LIN {X 0,Y 505.986,Z 301.18,A -85,B 0,C 180,E1 23907.931,E2 23907.931} C_VEL
LIN {X 0,Y 499.705,Z 283.022,A -85,B 0,C 180,E1 23905.729,E2 23905.729} C_VEL
LIN {X 0,Y 496.793,Z 274.791,A -85,B 0,C 180,E1 23904.638,E2 23904.638} C_VEL
LIN {X 0,Y 496.772,Z 274.605,A -85,B 0,C 180,E1 23901.099,E2 23901.099} C_VEL
LIN {X 0,Y 496.748,Z 274.605,A -85,B 0,C 180,E1 23897.6,E2 23897.6} C_VEL
LIN {X 0,Y 496.751,Z 274.607,A -85,B 0,C 180,E1 23893.982,E2 23893.982} C_VEL
LIN {X 0,Y 496.769,Z 274.603,A -85,B 0,C 180,E1 23890.399,E2 23890.399} C_VEL
LIN {X 0,Y 496.757,Z 274.604,A -85,B 0,C 180,E1 23886.857,E2 23886.857} C_VEL
LIN {X 0,Y 496.761,Z 274.607,A -85,B 0,C 180,E1 23883.333,E2 23883.333} C_VEL
LIN {X 0,Y 496.769,Z 274.598,A -85,B 0,C 180,E1 23879.812,E2 23879.812} C_VEL
LIN {X 0,Y 496.768,Z 274.604,A -85,B 0,C 180,E1 23876.284,E2 23876.284} C_VEL
LIN {X 0,Y 496.734,Z 274.607,A -85,B 0,C 180,E1 23872.794,E2 23872.794} C_VEL
LIN {X 0,Y 496.727,Z 274.609,A -85,B 0,C 180,E1 23869.255,E2 23869.255} C_VEL
LIN {X 0,Y 496.753,Z 274.6,A -85,B 0,C 180,E1 23865.768,E2 23865.768} C_VEL
LIN {X 0,Y 496.743,Z 274.605,A -85,B 0,C 180,E1 23862.32,E2 23862.32} C_VEL
LIN {X 0,Y 496.744,Z 274.899,A -85,B 0,C 180,E1 23861.172,E2 23861.172} C_VEL
LIN {X 0,Y 503.539,Z 295.552,A -85,B 0,C 180,E1 23858.969,E2 23858.969} C_VEL
LIN {X 0,Y 503.974,Z 298.794,A -85,B 0,C 180,E1 23858.673,E2 23858.673} C_VEL
LIN {X 0,Y 503.208,Z 340.602,A -85,B 0,C 180,E1 23855.245,E2 23855.245} C_VEL
LIN {X 0,Y 502.249,Z 380.984,A -85,B 0,C 180,E1 23851.941,E2 23851.941} C_VEL
LIN {X 0,Y 501.067,Z 425.768,A -85,B 0,C 180,E1 23848.286,E2 23848.286} C_VEL
LIN {X 0,Y 500.006,Z 468.043,A -85,B 0,C 180,E1 23844.839,E2 23844.839} C_VEL
LIN {X 0,Y 499.903,Z 474.861,A -85,B 0,C 180,E1 23844.316,E2 23844.316} C_VEL
LIN {X 0,Y 500.969,Z 485.924,A -85,B 0,C 180,E1 23844.105,E2 23844.105} C_VEL
LIN {X 0,Y 499.941,Z 617.34,A -85,B 0,C 180,E1 23842.16,E2 23842.16} C_VEL
LIN {X 0,Y 499.655,Z 633.277,A -85,B 0,C 180,E1 23841.714,E2 23841.714} C_VEL
LIN {X 0,Y 499.205,Z 649.81,A -85,B 0,C 180,E1 23841.013,E2 23841.013} C_VEL
LIN {X 0,Y 498.696,Z 664.017,A -85,B 0,C 180,E1 23840.189,E2 23840.189} C_VEL
LIN {X 0,Y 498.107,Z 678.224,A -85,B 0,C 180,E1 23839.125,E2 23839.125} C_VEL
LIN {X 0,Y 497.578,Z 690.76,A -85,B 0,C 180,E1 23837.939,E2 23837.939} C_VEL
LIN {X 0,Y 497.048,Z 702.83,A -85,B 0,C 180,E1 23836.507,E2 23836.507} C_VEL
LIN {X 0,Y 496.653,Z 712.568,A -85,B 0,C 180,E1 23835.069,E2 23835.069} C_VEL
LIN {X 0,Y 496.323,Z 721.598,A -85,B 0,C 180,E1 23833.379,E2 23833.379} C_VEL
LIN {X 0,Y 496.123,Z 728.676,A -85,B 0,C 180,E1 23831.666,E2 23831.666} C_VEL
LIN {X 0,Y 496.01,Z 734.174,A -85,B 0,C 180,E1 23829.838,E2 23829.838} C_VEL
LIN {X 0,Y 495.963,Z 737.914,A -85,B 0,C 180,E1 23827.979,E2 23827.979} C_VEL
LIN {X 0,Y 495.946,Z 739.841,A -85,B 0,C 180,E1 23826.096,E2 23826.096} C_VEL
LIN {X 0,Y 495.945,Z 740.052,A -85,B 0,C 180,E1 23824.187,E2 23824.187} C_VEL
LIN {X 0,Y 495.956,Z 738.355,A -85,B 0,C 180,E1 23822.246,E2 23822.246} C_VEL
LIN {X 0,Y 496.004,Z 734.845,A -85,B 0,C 180,E1 23820.323,E2 23820.323} C_VEL
LIN {X 0,Y 496.106,Z 729.548,A -85,B 0,C 180,E1 23818.488,E2 23818.488} C_VEL
LIN {X 0,Y 496.302,Z 722.599,A -85,B 0,C 180,E1 23816.728,E2 23816.728} C_VEL
LIN {X 0,Y 496.624,Z 713.491,A -85,B 0,C 180,E1 23814.987,E2 23814.987} C_VEL
LIN {X 0,Y 497.041,Z 703.344,A -85,B 0,C 180,E1 23813.458,E2 23813.458} C_VEL
LIN {X 0,Y 497.549,Z 691.637,A -85,B 0,C 180,E1 23812.056,E2 23812.056} C_VEL
LIN {X 0,Y 498.077,Z 679.489,A -85,B 0,C 180,E1 23810.881,E2 23810.881} C_VEL
LIN {X 0,Y 498.659,Z 665.144,A -85,B 0,C 180,E1 23809.789,E2 23809.789} C_VEL
LIN {X 0,Y 499.193,Z 650.674,A -85,B 0,C 180,E1 23808.933,E2 23808.933} C_VEL
LIN {X 0,Y 499.631,Z 634.514,A -85,B 0,C 180,E1 23808.237,E2 23808.237} C_VEL
LIN {X 0,Y 499.922,Z 618.388,A -85,B 0,C 180,E1 23807.769,E2 23807.769} C_VEL
LIN {X 0,Y 500.3,Z 568.29,A -85,B 0,C 180,E1 23807.005,E2 23807.005} C_VEL
LIN {X 0,Y 500.781,Z 482.143,A -85,B 0,C 180,E1 23805.739,E2 23805.739} C_VEL
LIN {X 0,Y 499.842,Z 474.397,A -85,B 0,C 180,E1 23805.566,E2 23805.566} C_VEL
LIN {X 0,Y 500.963,Z 429.094,A -85,B 0,C 180,E1 23801.89,E2 23801.89} C_VEL
LIN {X 0,Y 501.829,Z 393.421,A -85,B 0,C 180,E1 23799.012,E2 23799.012} C_VEL
LIN {X 0,Y 502.557,Z 361.365,A -85,B 0,C 180,E1 23796.433,E2 23796.433} C_VEL
LIN {X 0,Y 503.208,Z 320.138,A -85,B 0,C 180,E1 23793.122,E2 23793.122} C_VEL
LIN {X 0,Y 503.4,Z 295.62,A -85,B 0,C 180,E1 23791.159,E2 23791.159} C_VEL
LIN {X 0,Y 496.791,Z 274.932,A -85,B 0,C 180,E1 23789.049,E2 23789.049} C_VEL
LIN {X 0,Y 496.729,Z 274.611,A -85,B 0,C 180,E1 23788.363,E2 23788.363} C_VEL
LIN {X 0,Y 496.731,Z 274.611,A -85,B 0,C 180,E1 23784.752,E2 23784.752} C_VEL
LIN {X 0,Y 496.766,Z 274.602,A -85,B 0,C 180,E1 23781.242,E2 23781.242} C_VEL
LIN {X 0,Y 496.764,Z 274.605,A -85,B 0,C 180,E1 23777.694,E2 23777.694} C_VEL
LIN {X 0,Y 496.729,Z 274.608,A -85,B 0,C 180,E1 23774.216,E2 23774.216} C_VEL
LIN {X 0,Y 496.736,Z 274.605,A -85,B 0,C 180,E1 23770.672,E2 23770.672} C_VEL
LIN {X 0,Y 496.774,Z 274.603,A -85,B 0,C 180,E1 23767.148,E2 23767.148} C_VEL
LIN {X 0,Y 496.764,Z 274.607,A -85,B 0,C 180,E1 23763.578,E2 23763.578} C_VEL
LIN {X 0,Y 496.733,Z 274.608,A -85,B 0,C 180,E1 23760.116,E2 23760.116} C_VEL
LIN {X 0,Y 496.738,Z 274.604,A -85,B 0,C 180,E1 23756.538,E2 23756.538} C_VEL
LIN {X 0,Y 496.773,Z 274.603,A -85,B 0,C 180,E1 23753.064,E2 23753.064} C_VEL
LIN {X 0,Y 496.757,Z 274.606,A -85,B 0,C 180,E1 23749.564,E2 23749.564} C_VEL
LIN {X 0,Y 496.734,Z 274.606,A -85,B 0,C 180,E1 23746.023,E2 23746.023} C_VEL
LIN {X 0,Y 496.744,Z 274.605,A -85,B 0,C 180,E1 23742.427,E2 23742.427} C_VEL
LIN {X 0,Y 496.771,Z 274.602,A -85,B 0,C 180,E1 23738.883,E2 23738.883} C_VEL
LIN {X 0,Y 496.763,Z 274.607,A -85,B 0,C 180,E1 23735.378,E2 23735.378} C_VEL
LIN {X 0,Y 496.738,Z 274.607,A -85,B 0,C 180,E1 23731.835,E2 23731.835} C_VEL
LIN {X 0,Y 496.746,Z 274.603,A -85,B 0,C 180,E1 23728.309,E2 23728.309} C_VEL
LIN {X 0,Y 496.772,Z 274.604,A -85,B 0,C 180,E1 23724.798,E2 23724.798} C_VEL
LIN {X 0,Y 496.767,Z 274.609,A -85,B 0,C 180,E1 23721.248,E2 23721.248} C_VEL
LIN {X 0,Y 496.739,Z 274.609,A -85,B 0,C 180,E1 23717.756,E2 23717.756} C_VEL
LIN {X 0,Y 496.751,Z 274.605,A -85,B 0,C 180,E1 23714.23,E2 23714.23} C_VEL
LIN {X 0,Y 496.772,Z 274.607,A -85,B 0,C 180,E1 23710.699,E2 23710.699} C_VEL
LIN {X 0,Y 496.777,Z 274.865,A -85,B 0,C 180,E1 23707.944,E2 23707.944} C_VEL
LIN {X 0,Y 500.523,Z 284.291,A -85,B 0,C 180,E1 23706.77,E2 23706.77} C_VEL
LIN {X 0,Y 508.094,Z 303.988,A -85,B 0,C 180,E1 23704.559,E2 23704.559} C_VEL
LIN {X 0,Y 507.57,Z 316.675,A -85,B 0,C 180,E1 23703.616,E2 23703.616} C_VEL
LIN {X 0,Y 510.176,Z 334.45,A -85,B 0,C 180,E1 23703.112,E2 23703.112} C_VEL
LIN {X 0,Y 508.469,Z 453.813,A -85,B 0,C 180,E1 23701.237,E2 23701.237} C_VEL
LIN {X 0,Y 506.934,Z 577.933,A -85,B 0,C 180,E1 23699.32,E2 23699.32} C_VEL
LIN {X 0,Y 506.225,Z 599.572,A -85,B 0,C 180,E1 23698.769,E2 23698.769} C_VEL
LIN {X 0,Y 505.38,Z 619.891,A -85,B 0,C 180,E1 23698.031,E2 23698.031} C_VEL
LIN {X 0,Y 504.378,Z 639.254,A -85,B 0,C 180,E1 23697.117,E2 23697.117} C_VEL
LIN {X 0,Y 503.262,Z 658.557,A -85,B 0,C 180,E1 23695.981,E2 23695.981} C_VEL
LIN {X 0,Y 502.09,Z 677.202,A -85,B 0,C 180,E1 23694.641,E2 23694.641} C_VEL
LIN {X 0,Y 500.925,Z 694.485,A -85,B 0,C 180,E1 23693.153,E2 23693.153} C_VEL
LIN {X 0,Y 499.847,Z 710.302,A -85,B 0,C 180,E1 23691.542,E2 23691.542} C_VEL
LIN {X 0,Y 498.832,Z 724.453,A -85,B 0,C 180,E1 23689.799,E2 23689.799} C_VEL
LIN {X 0,Y 497.924,Z 737.789,A -85,B 0,C 180,E1 23687.859,E2 23687.859} C_VEL
LIN {X 0,Y 497.213,Z 749.382,A -85,B 0,C 180,E1 23685.87,E2 23685.87} C_VEL
LIN {X 0,Y 496.65,Z 760.337,A -85,B 0,C 180,E1 23683.622,E2 23683.622} C_VEL
LIN {X 0,Y 496.279,Z 769.255,A -85,B 0,C 180,E1 23681.386,E2 23681.386} C_VEL
LIN {X 0,Y 496.067,Z 776.378,A -85,B 0,C 180,E1 23679.161,E2 23679.161} C_VEL
LIN {X 0,Y 495.965,Z 782.008,A -85,B 0,C 180,E1 23676.83,E2 23676.83} C_VEL
LIN {X 0,Y 495.918,Z 785.929,A -85,B 0,C 180,E1 23674.509,E2 23674.509} C_VEL
LIN {X 0,Y 495.911,Z 788.305,A -85,B 0,C 180,E1 23672.079,E2 23672.079} C_VEL
LIN {X 0,Y 495.906,Z 788.962,A -85,B 0,C 180,E1 23669.768,E2 23669.768} C_VEL
LIN {X 0,Y 495.908,Z 788.03,A -85,B 0,C 180,E1 23667.456,E2 23667.456} C_VEL
LIN {X 0,Y 495.924,Z 785.445,A -85,B 0,C 180,E1 23665.141,E2 23665.141} C_VEL
LIN {X 0,Y 495.964,Z 781.241,A -85,B 0,C 180,E1 23662.819,E2 23662.819} C_VEL
LIN {X 0,Y 496.095,Z 775.322,A -85,B 0,C 180,E1 23660.486,E2 23660.486} C_VEL
LIN {X 0,Y 496.335,Z 767.956,A -85,B 0,C 180,E1 23658.247,E2 23658.247} C_VEL
LIN {X 0,Y 496.733,Z 758.589,A -85,B 0,C 180,E1 23655.977,E2 23655.977} C_VEL
LIN {X 0,Y 497.288,Z 748.099,A -85,B 0,C 180,E1 23653.89,E2 23653.89} C_VEL
LIN {X 0,Y 498.033,Z 736.03,A -85,B 0,C 180,E1 23651.869,E2 23651.869} C_VEL
LIN {X 0,Y 499.023,Z 721.655,A -85,B 0,C 180,E1 23649.84,E2 23649.84} C_VEL
LIN {X 0,Y 500.037,Z 707.603,A -85,B 0,C 180,E1 23648.165,E2 23648.165} C_VEL
LIN {X 0,Y 501.074,Z 691.666,A -85,B 0,C 180,E1 23646.603,E2 23646.603} C_VEL
LIN {X 0,Y 502.192,Z 674.015,A -85,B 0,C 180,E1 23645.158,E2 23645.158} C_VEL
LIN {X 0,Y 503.256,Z 655.481,A -85,B 0,C 180,E1 23643.899,E2 23643.899} C_VEL
LIN {X 0,Y 504.197,Z 636.876,A -85,B 0,C 180,E1 23642.863,E2 23642.863} C_VEL
LIN {X 0,Y 505.11,Z 616.417,A -85,B 0,C 180,E1 23641.956,E2 23641.956} C_VEL
LIN {X 0,Y 505.853,Z 595.464,A -85,B 0,C 180,E1 23641.258,E2 23641.258} C_VEL
LIN {X 0,Y 506.394,Z 574.481,A -85,B 0,C 180,E1 23640.774,E2 23640.774} C_VEL
LIN {X 0,Y 508.288,Z 392.914,A -85,B 0,C 180,E1 23638.038,E2 23638.038} C_VEL
LIN {X 0,Y 509.019,Z 331.819,A -85,B 0,C 180,E1 23637.033,E2 23637.033} C_VEL
LIN {X 0,Y 506.9,Z 317.552,A -85,B 0,C 180,E1 23636.61,E2 23636.61} C_VEL
LIN {X 0,Y 507.597,Z 303.416,A -85,B 0,C 180,E1 23635.523,E2 23635.523} C_VEL
LIN {X 0,Y 501.679,Z 286.882,A -85,B 0,C 180,E1 23633.563,E2 23633.563} C_VEL
LIN {X 0,Y 498.35,Z 278.58,A -85,B 0,C 180,E1 23632.415,E2 23632.415} C_VEL
LIN {X 0,Y 496.787,Z 274.85,A -85,B 0,C 180,E1 23631.796,E2 23631.796} C_VEL
LIN {X 0,Y 496.734,Z 274.612,A -85,B 0,C 180,E1 23628.311,E2 23628.311} C_VEL
LIN {X 0,Y 496.754,Z 274.611,A -85,B 0,C 180,E1 23624.787,E2 23624.787} C_VEL
LIN {X 0,Y 496.775,Z 274.607,A -85,B 0,C 180,E1 23621.312,E2 23621.312} C_VEL
LIN {X 0,Y 496.735,Z 274.612,A -85,B 0,C 180,E1 23617.873,E2 23617.873} C_VEL
LIN {X 0,Y 496.768,Z 274.901,A -85,B 0,C 180,E1 23616.1,E2 23616.1} C_VEL
LIN {X 0,Y 500.068,Z 282.968,A -85,B 0,C 180,E1 23614.736,E2 23614.736} C_VEL
LIN {X 0,Y 504.417,Z 294.778,A -85,B 0,C 180,E1 23613.032,E2 23613.032} C_VEL
LIN {X 0,Y 506.659,Z 302.39,A -85,B 0,C 180,E1 23612.063,E2 23612.063} C_VEL
LIN {X 0,Y 504.302,Z 341.082,A -85,B 0,C 180,E1 23608.577,E2 23608.577} C_VEL
LIN {X 0,Y 507.189,Z 359.883,A -85,B 0,C 180,E1 23608.008,E2 23608.008} C_VEL
LIN {X 0,Y 505.208,Z 474.152,A -85,B 0,C 180,E1 23606.152,E2 23606.152} C_VEL
LIN {X 0,Y 504.179,Z 561.011,A -85,B 0,C 180,E1 23604.803,E2 23604.803} C_VEL
LIN {X 0,Y 503.6,Z 581.084,A -85,B 0,C 180,E1 23604.273,E2 23604.273} C_VEL
LIN {X 0,Y 502.863,Z 599.834,A -85,B 0,C 180,E1 23603.556,E2 23603.556} C_VEL
LIN {X 0,Y 501.968,Z 618.446,A -85,B 0,C 180,E1 23602.608,E2 23602.608} C_VEL
LIN {X 0,Y 501.011,Z 635.928,A -85,B 0,C 180,E1 23601.482,E2 23601.482} C_VEL
LIN {X 0,Y 500.015,Z 652.165,A -85,B 0,C 180,E1 23600.178,E2 23600.178} C_VEL
LIN {X 0,Y 498.991,Z 668.376,A -85,B 0,C 180,E1 23598.596,E2 23598.596} C_VEL
LIN {X 0,Y 498.163,Z 681.6,A -85,B 0,C 180,E1 23597.039,E2 23597.039} C_VEL
LIN {X 0,Y 497.426,Z 694.289,A -85,B 0,C 180,E1 23595.267,E2 23595.267} C_VEL
LIN {X 0,Y 496.85,Z 705.515,A -85,B 0,C 180,E1 23593.381,E2 23593.381} C_VEL
LIN {X 0,Y 496.427,Z 715.203,A -85,B 0,C 180,E1 23591.384,E2 23591.384} C_VEL
LIN {X 0,Y 496.162,Z 722.983,A -85,B 0,C 180,E1 23589.394,E2 23589.394} C_VEL
LIN {X 0,Y 496.006,Z 729.436,A -85,B 0,C 180,E1 23587.296,E2 23587.296} C_VEL
LIN {X 0,Y 495.94,Z 734.373,A -85,B 0,C 180,E1 23585.089,E2 23585.089} C_VEL
LIN {X 0,Y 495.914,Z 737.458,A -85,B 0,C 180,E1 23582.889,E2 23582.889} C_VEL
LIN {X 0,Y 495.914,Z 738.85,A -85,B 0,C 180,E1 23580.693,E2 23580.693} C_VEL
LIN {X 0,Y 495.91,Z 738.609,A -85,B 0,C 180,E1 23578.498,E2 23578.498} C_VEL
LIN {X 0,Y 495.912,Z 736.657,A -85,B 0,C 180,E1 23576.3,E2 23576.3} C_VEL
LIN {X 0,Y 495.949,Z 732.923,A -85,B 0,C 180,E1 23574.098,E2 23574.098} C_VEL
LIN {X 0,Y 496.049,Z 727.391,A -85,B 0,C 180,E1 23571.888,E2 23571.888} C_VEL
LIN {X 0,Y 496.238,Z 720.359,A -85,B 0,C 180,E1 23569.786,E2 23569.786} C_VEL
LIN {X 0,Y 496.56,Z 711.892,A -85,B 0,C 180,E1 23567.794,E2 23567.794} C_VEL
LIN {X 0,Y 497.034,Z 701.633,A -85,B 0,C 180,E1 23565.842,E2 23565.842} C_VEL
LIN {X 0,Y 497.658,Z 690.096,A -85,B 0,C 180,E1 23564.023,E2 23564.023} C_VEL
LIN {X 0,Y 498.427,Z 677.376,A -85,B 0,C 180,E1 23562.34,E2 23562.34} C_VEL
LIN {X 0,Y 499.319,Z 663.137,A -85,B 0,C 180,E1 23560.767,E2 23560.767} C_VEL
LIN {X 0,Y 500.335,Z 646.924,A -85,B 0,C 180,E1 23559.285,E2 23559.285} C_VEL
LIN {X 0,Y 501.337,Z 630.264,A -85,B 0,C 180,E1 23558.033,E2 23558.033} C_VEL
LIN {X 0,Y 502.287,Z 612.613,A -85,B 0,C 180,E1 23556.973,E2 23556.973} C_VEL
LIN {X 0,Y 503.176,Z 593.403,A -85,B 0,C 180,E1 23556.074,E2 23556.074} C_VEL
LIN {X 0,Y 503.874,Z 574.138,A -85,B 0,C 180,E1 23555.411,E2 23555.411} C_VEL
LIN {X 0,Y 504.363,Z 554.443,A -85,B 0,C 180,E1 23554.966,E2 23554.966} C_VEL
LIN {X 0,Y 506.641,Z 358.228,A -85,B 0,C 180,E1 23551.968,E2 23551.968} C_VEL
LIN {X 0,Y 505.059,Z 353.42,A -85,B 0,C 180,E1 23551.781,E2 23551.781} C_VEL
LIN {X 0,Y 499.919,Z 345.851,A -85,B 0,C 180,E1 23551.315,E2 23551.315} C_VEL
LIN {X 0,Y 497.214,Z 341.288,A -85,B 0,C 180,E1 23550.985,E2 23550.985} C_VEL
LIN {X 0,Y 496.832,Z 338.92,A -85,B 0,C 180,E1 23550.787,E2 23550.787} C_VEL
LIN {X 0,Y 498.75,Z 303.753,A -85,B 0,C 180,E1 23547.638,E2 23547.638} C_VEL
LIN {X 0,Y 491.879,Z 284.216,A -85,B 0,C 180,E1 23545.209,E2 23545.209} C_VEL
LIN {X 0,Y 488.822,Z 275.791,A -85,B 0,C 180,E1 23544.059,E2 23544.059} C_VEL
LIN {X 0,Y 488.834,Z 275.59,A -85,B 0,C 180,E1 23540.64,E2 23540.64} C_VEL
LIN {X 0,Y 488.83,Z 275.597,A -85,B 0,C 180,E1 23537.068,E2 23537.068} C_VEL
LIN {X 0,Y 488.823,Z 275.593,A -85,B 0,C 180,E1 23533.436,E2 23533.436} C_VEL
LIN {X 0,Y 488.818,Z 275.596,A -85,B 0,C 180,E1 23529.91,E2 23529.91} C_VEL
LIN {X 0,Y 488.828,Z 275.591,A -85,B 0,C 180,E1 23526.302,E2 23526.302} C_VEL
LIN {X 0,Y 488.814,Z 275.593,A -85,B 0,C 180,E1 23522.786,E2 23522.786} C_VEL
LIN {X 0,Y 488.806,Z 275.588,A -85,B 0,C 180,E1 23519.134,E2 23519.134} C_VEL
LIN {X 0,Y 488.82,Z 275.588,A -85,B 0,C 180,E1 23515.57,E2 23515.57} C_VEL
LIN {X 0,Y 488.836,Z 275.591,A -85,B 0,C 180,E1 23511.982,E2 23511.982} C_VEL
LIN {X 0,Y 488.804,Z 275.594,A -85,B 0,C 180,E1 23508.486,E2 23508.486} C_VEL
LIN {X 0,Y 488.771,Z 275.58,A -85,B 0,C 180,E1 23505.059,E2 23505.059} C_VEL
LIN {X 0,Y 488.803,Z 275.676,A -85,B 0,C 180,E1 23501.685,E2 23501.685} C_VEL
LIN {X 0,Y 489.195,Z 277.342,A -85,B 0,C 180,E1 23501.436,E2 23501.436} C_VEL
LIN {X 0,Y 495.993,Z 297.471,A -85,B 0,C 180,E1 23499.282,E2 23499.282} C_VEL
LIN {X 0,Y 496.654,Z 300.627,A -85,B 0,C 180,E1 23498.977,E2 23498.977} C_VEL
LIN {X 0,Y 495.796,Z 341.958,A -85,B 0,C 180,E1 23495.556,E2 23495.556} C_VEL
LIN {X 0,Y 494.775,Z 382.728,A -85,B 0,C 180,E1 23492.202,E2 23492.202} C_VEL
LIN {X 0,Y 493.521,Z 426.283,A -85,B 0,C 180,E1 23488.608,E2 23488.608} C_VEL
LIN {X 0,Y 492.405,Z 467.332,A -85,B 0,C 180,E1 23485.226,E2 23485.226} C_VEL
LIN {X 0,Y 492.302,Z 475.276,A -85,B 0,C 180,E1 23484.622,E2 23484.622} C_VEL
LIN {X 0,Y 493.414,Z 486.66,A -85,B 0,C 180,E1 23484.401,E2 23484.401} C_VEL
LIN {X 0,Y 492.302,Z 617.759,A -85,B 0,C 180,E1 23482.43,E2 23482.43} C_VEL
LIN {X 0,Y 491.997,Z 633.675,A -85,B 0,C 180,E1 23481.977,E2 23481.977} C_VEL
LIN {X 0,Y 491.529,Z 649.708,A -85,B 0,C 180,E1 23481.291,E2 23481.291} C_VEL
LIN {X 0,Y 490.98,Z 664.147,A -85,B 0,C 180,E1 23480.448,E2 23480.448} C_VEL
LIN {X 0,Y 490.347,Z 678.333,A -85,B 0,C 180,E1 23479.373,E2 23479.373} C_VEL
LIN {X 0,Y 489.798,Z 690.444,A -85,B 0,C 180,E1 23478.222,E2 23478.222} C_VEL
LIN {X 0,Y 489.211,Z 702.633,A -85,B 0,C 180,E1 23476.769,E2 23476.769} C_VEL
LIN {X 0,Y 488.771,Z 712.504,A -85,B 0,C 180,E1 23475.307,E2 23475.307} C_VEL
LIN {X 0,Y 488.399,Z 721.62,A -85,B 0,C 180,E1 23473.591,E2 23473.591} C_VEL
LIN {X 0,Y 488.172,Z 728.757,A -85,B 0,C 180,E1 23471.863,E2 23471.863} C_VEL
LIN {X 0,Y 488.035,Z 734.364,A -85,B 0,C 180,E1 23469.994,E2 23469.994} C_VEL
LIN {X 0,Y 487.976,Z 738.186,A -85,B 0,C 180,E1 23468.106,E2 23468.106} C_VEL
LIN {X 0,Y 487.956,Z 740.184,A -85,B 0,C 180,E1 23466.194,E2 23466.194} C_VEL
LIN {X 0,Y 487.954,Z 740.463,A -85,B 0,C 180,E1 23464.254,E2 23464.254} C_VEL
LIN {X 0,Y 487.967,Z 739.029,A -85,B 0,C 180,E1 23462.416,E2 23462.416} C_VEL
LIN {X 0,Y 488.015,Z 735.602,A -85,B 0,C 180,E1 23460.413,E2 23460.413} C_VEL
LIN {X 0,Y 488.119,Z 730.832,A -85,B 0,C 180,E1 23458.65,E2 23458.65} C_VEL
LIN {X 0,Y 488.321,Z 724.137,A -85,B 0,C 180,E1 23456.861,E2 23456.861} C_VEL
LIN {X 0,Y 488.636,Z 715.973,A -85,B 0,C 180,E1 23455.189,E2 23455.189} C_VEL
LIN {X 0,Y 489.088,Z 705.62,A -85,B 0,C 180,E1 23453.537,E2 23453.537} C_VEL
LIN {X 0,Y 489.608,Z 694.729,A -85,B 0,C 180,E1 23452.147,E2 23452.147} C_VEL
LIN {X 0,Y 490.22,Z 681.581,A -85,B 0,C 180,E1 23450.811,E2 23450.811} C_VEL
LIN {X 0,Y 490.835,Z 668.041,A -85,B 0,C 180,E1 23449.72,E2 23449.72} C_VEL
LIN {X 0,Y 491.443,Z 652.629,A -85,B 0,C 180,E1 23448.764,E2 23448.764} C_VEL
LIN {X 0,Y 491.923,Z 637.265,A -85,B 0,C 180,E1 23448.061,E2 23448.061} C_VEL
LIN {X 0,Y 492.26,Z 620.466,A -85,B 0,C 180,E1 23447.538,E2 23447.538} C_VEL
LIN {X 0,Y 492.473,Z 597.604,A -85,B 0,C 180,E1 23447.149,E2 23447.149} C_VEL
LIN {X 0,Y 493.242,Z 483.022,A -85,B 0,C 180,E1 23445.442,E2 23445.442} C_VEL
LIN {X 0,Y 492.238,Z 474.376,A -85,B 0,C 180,E1 23445.229,E2 23445.229} C_VEL
LIN {X 0,Y 493.397,Z 430.05,A -85,B 0,C 180,E1 23441.605,E2 23441.605} C_VEL
LIN {X 0,Y 494.609,Z 387.909,A -85,B 0,C 180,E1 23438.156,E2 23438.156} C_VEL
LIN {X 0,Y 495.441,Z 344.839,A -85,B 0,C 180,E1 23434.689,E2 23434.689} C_VEL
LIN {X 0,Y 496.02,Z 306.668,A -85,B 0,C 180,E1 23431.608,E2 23431.608} C_VEL
LIN {X 0,Y 495.9,Z 297.676,A -85,B 0,C 180,E1 23430.874,E2 23430.874} C_VEL
LIN {X 0,Y 489.365,Z 277.73,A -85,B 0,C 180,E1 23428.829,E2 23428.829} C_VEL
LIN {X 0,Y 488.811,Z 275.772,A -85,B 0,C 180,E1 23428.567,E2 23428.567} C_VEL
LIN {X 0,Y 488.819,Z 275.596,A -85,B 0,C 180,E1 23425.18,E2 23425.18} C_VEL
LIN {X 0,Y 488.834,Z 275.592,A -85,B 0,C 180,E1 23421.603,E2 23421.603} C_VEL
LIN {X 0,Y 488.797,Z 275.593,A -85,B 0,C 180,E1 23418.115,E2 23418.115} C_VEL
LIN {X 0,Y 488.79,Z 275.595,A -85,B 0,C 180,E1 23414.573,E2 23414.573} C_VEL
LIN {X 0,Y 488.823,Z 275.593,A -85,B 0,C 180,E1 23411.086,E2 23411.086} C_VEL
LIN {X 0,Y 488.834,Z 275.597,A -85,B 0,C 180,E1 23407.522,E2 23407.522} C_VEL
LIN {X 0,Y 488.799,Z 275.597,A -85,B 0,C 180,E1 23403.988,E2 23403.988} C_VEL
LIN {X 0,Y 488.793,Z 275.596,A -85,B 0,C 180,E1 23400.352,E2 23400.352} C_VEL
LIN {X 0,Y 488.817,Z 275.592,A -85,B 0,C 180,E1 23396.834,E2 23396.834} C_VEL
LIN {X 0,Y 488.833,Z 275.593,A -85,B 0,C 180,E1 23393.305,E2 23393.305} C_VEL
LIN {X 0,Y 488.806,Z 275.594,A -85,B 0,C 180,E1 23389.749,E2 23389.749} C_VEL
LIN {X 0,Y 488.794,Z 275.595,A -85,B 0,C 180,E1 23386.153,E2 23386.153} C_VEL
LIN {X 0,Y 488.816,Z 275.593,A -85,B 0,C 180,E1 23382.625,E2 23382.625} C_VEL
LIN {X 0,Y 488.835,Z 275.592,A -85,B 0,C 180,E1 23379.026,E2 23379.026} C_VEL
LIN {X 0,Y 488.819,Z 275.597,A -85,B 0,C 180,E1 23375.467,E2 23375.467} C_VEL
LIN {X 0,Y 488.797,Z 275.595,A -85,B 0,C 180,E1 23371.935,E2 23371.935} C_VEL
LIN {X 0,Y 488.814,Z 275.592,A -85,B 0,C 180,E1 23368.423,E2 23368.423} C_VEL
LIN {X 0,Y 488.833,Z 275.594,A -85,B 0,C 180,E1 23364.898,E2 23364.898} C_VEL
LIN {X 0,Y 488.828,Z 275.598,A -85,B 0,C 180,E1 23361.252,E2 23361.252} C_VEL
LIN {X 0,Y 488.802,Z 275.598,A -85,B 0,C 180,E1 23357.703,E2 23357.703} C_VEL
LIN {X 0,Y 488.806,Z 275.595,A -85,B 0,C 180,E1 23354.063,E2 23354.063} C_VEL
LIN {X 0,Y 488.832,Z 275.595,A -85,B 0,C 180,E1 23350.458,E2 23350.458} C_VEL
LIN {X 0,Y 488.869,Z 275.852,A -85,B 0,C 180,E1 23348.554,E2 23348.554} C_VEL
LIN {X 0,Y 492.109,Z 284.143,A -85,B 0,C 180,E1 23347.495,E2 23347.495} C_VEL
LIN {X 0,Y 500.017,Z 304.476,A -85,B 0,C 180,E1 23345.13,E2 23345.13} C_VEL
LIN {X 0,Y 500.977,Z 307.529,A -85,B 0,C 180,E1 23344.804,E2 23344.804} C_VEL
LIN {X 0,Y 500.587,Z 316.917,A -85,B 0,C 180,E1 23344.109,E2 23344.109} C_VEL
LIN {X 0,Y 503.315,Z 335.797,A -85,B 0,C 180,E1 23343.562,E2 23343.562} C_VEL
LIN {X 0,Y 501.332,Z 459.092,A -85,B 0,C 180,E1 23341.584,E2 23341.584} C_VEL
LIN {X 0,Y 499.699,Z 577.734,A -85,B 0,C 180,E1 23339.715,E2 23339.715} C_VEL
LIN {X 0,Y 498.941,Z 599.291,A -85,B 0,C 180,E1 23339.159,E2 23339.159} C_VEL
LIN {X 0,Y 498.031,Z 619.627,A -85,B 0,C 180,E1 23338.41,E2 23338.41} C_VEL
LIN {X 0,Y 496.93,Z 639.428,A -85,B 0,C 180,E1 23337.462,E2 23337.462} C_VEL
LIN {X 0,Y 495.733,Z 658.737,A -85,B 0,C 180,E1 23336.303,E2 23336.303} C_VEL
LIN {X 0,Y 494.467,Z 677.403,A -85,B 0,C 180,E1 23334.936,E2 23334.936} C_VEL
LIN {X 0,Y 493.206,Z 694.771,A -85,B 0,C 180,E1 23333.41,E2 23333.41} C_VEL
LIN {X 0,Y 492.068,Z 710.441,A -85,B 0,C 180,E1 23331.783,E2 23331.783} C_VEL
LIN {X 0,Y 491.027,Z 725.018,A -85,B 0,C 180,E1 23330.003,E2 23330.003} C_VEL
LIN {X 0,Y 490.151,Z 737.581,A -85,B 0,C 180,E1 23328.184,E2 23328.184} C_VEL
LIN {X 0,Y 489.358,Z 749.381,A -85,B 0,C 180,E1 23326.132,E2 23326.132} C_VEL
LIN {X 0,Y 488.733,Z 760.337,A -85,B 0,C 180,E1 23323.847,E2 23323.847} C_VEL
LIN {X 0,Y 488.326,Z 769.254,A -85,B 0,C 180,E1 23321.574,E2 23321.574} C_VEL
LIN {X 0,Y 488.086,Z 776.378,A -85,B 0,C 180,E1 23319.312,E2 23319.312} C_VEL
LIN {X 0,Y 487.968,Z 782.008,A -85,B 0,C 180,E1 23316.942,E2 23316.942} C_VEL
LIN {X 0,Y 487.919,Z 785.928,A -85,B 0,C 180,E1 23314.583,E2 23314.583} C_VEL
LIN {X 0,Y 487.91,Z 788.305,A -85,B 0,C 180,E1 23312.113,E2 23312.113} C_VEL
LIN {X 0,Y 487.906,Z 788.962,A -85,B 0,C 180,E1 23309.764,E2 23309.764} C_VEL
LIN {X 0,Y 487.909,Z 788.03,A -85,B 0,C 180,E1 23307.415,E2 23307.415} C_VEL
LIN {X 0,Y 487.924,Z 785.444,A -85,B 0,C 180,E1 23305.061,E2 23305.061} C_VEL
LIN {X 0,Y 487.972,Z 781.241,A -85,B 0,C 180,E1 23302.7,E2 23302.7} C_VEL
LIN {X 0,Y 488.119,Z 775.322,A -85,B 0,C 180,E1 23300.329,E2 23300.329} C_VEL
LIN {X 0,Y 488.381,Z 768.004,A -85,B 0,C 180,E1 23298.065,E2 23298.065} C_VEL
LIN {X 0,Y 488.815,Z 758.782,A -85,B 0,C 180,E1 23295.79,E2 23295.79} C_VEL
LIN {X 0,Y 489.44,Z 748.097,A -85,B 0,C 180,E1 23293.624,E2 23293.624} C_VEL
LIN {X 0,Y 490.254,Z 736.008,A -85,B 0,C 180,E1 23291.571,E2 23291.571} C_VEL
LIN {X 0,Y 491.139,Z 722.949,A -85,B 0,C 180,E1 23289.751,E2 23289.751} C_VEL
LIN {X 0,Y 492.149,Z 708.555,A -85,B 0,C 180,E1 23288.048,E2 23288.048} C_VEL
LIN {X 0,Y 493.292,Z 691.729,A -85,B 0,C 180,E1 23286.371,E2 23286.371} C_VEL
LIN {X 0,Y 494.425,Z 674.742,A -85,B 0,C 180,E1 23284.954,E2 23284.954} C_VEL
LIN {X 0,Y 495.528,Z 656.63,A -85,B 0,C 180,E1 23283.692,E2 23283.692} C_VEL
LIN {X 0,Y 496.623,Z 636.444,A -85,B 0,C 180,E1 23282.544,E2 23282.544} C_VEL
LIN {X 0,Y 497.584,Z 615.889,A -85,B 0,C 180,E1 23281.625,E2 23281.625} C_VEL
LIN {X 0,Y 498.379,Z 594.842,A -85,B 0,C 180,E1 23280.919,E2 23280.919} C_VEL
LIN {X 0,Y 498.936,Z 573.868,A -85,B 0,C 180,E1 23280.433,E2 23280.433} C_VEL
LIN {X 0,Y 500.822,Z 412.071,A -85,B 0,C 180,E1 23277.946,E2 23277.946} C_VEL
LIN {X 0,Y 502.027,Z 333.036,A -85,B 0,C 180,E1 23276.603,E2 23276.603} C_VEL
LIN {X 0,Y 499.908,Z 318.175,A -85,B 0,C 180,E1 23276.142,E2 23276.142} C_VEL
LIN {X 0,Y 500.482,Z 306.301,A -85,B 0,C 180,E1 23275.194,E2 23275.194} C_VEL
LIN {X 0,Y 495.135,Z 290.88,A -85,B 0,C 180,E1 23273.291,E2 23273.291} C_VEL
LIN {X 0,Y 491.749,Z 282.725,A -85,B 0,C 180,E1 23272.083,E2 23272.083} C_VEL
LIN {X 0,Y 489.923,Z 278.74,A -85,B 0,C 180,E1 23271.411,E2 23271.411} C_VEL
LIN {X 0,Y 488.841,Z 275.757,A -85,B 0,C 180,E1 23270.822,E2 23270.822} C_VEL
LIN {X 0,Y 488.834,Z 275.597,A -85,B 0,C 180,E1 23267.247,E2 23267.247} C_VEL
LIN {X 0,Y 488.81,Z 275.599,A -85,B 0,C 180,E1 23263.739,E2 23263.739} C_VEL
LIN {X 0,Y 488.79,Z 275.601,A -85,B 0,C 180,E1 23260.269,E2 23260.269} C_VEL
LIN {X 0,Y 488.863,Z 275.824,A -85,B 0,C 180,E1 23257.092,E2 23257.092} C_VEL
LIN {X 0,Y 490.357,Z 279.478,A -85,B 0,C 180,E1 23256.348,E2 23256.348} C_VEL
LIN {X 0,Y 493.795,Z 287.723,A -85,B 0,C 180,E1 23254.908,E2 23254.908} C_VEL
LIN {X 0,Y 497.768,Z 298.786,A -85,B 0,C 180,E1 23253.255,E2 23253.255} C_VEL
LIN {X 0,Y 499.736,Z 305.187,A -85,B 0,C 180,E1 23252.399,E2 23252.399} C_VEL
LIN {X 0,Y 497.286,Z 340.623,A -85,B 0,C 180,E1 23249.132,E2 23249.132} C_VEL
LIN {X 0,Y 500.347,Z 360.709,A -85,B 0,C 180,E1 23248.471,E2 23248.471} C_VEL
LIN {X 0,Y 497.85,Z 485.366,A -85,B 0,C 180,E1 23246.373,E2 23246.373} C_VEL
LIN {X 0,Y 496.774,Z 561.777,A -85,B 0,C 180,E1 23245.142,E2 23245.142} C_VEL
LIN {X 0,Y 496.153,Z 581.613,A -85,B 0,C 180,E1 23244.603,E2 23244.603} C_VEL
LIN {X 0,Y 495.386,Z 599.933,A -85,B 0,C 180,E1 23243.891,E2 23243.891} C_VEL
LIN {X 0,Y 494.481,Z 617.922,A -85,B 0,C 180,E1 23242.97,E2 23242.97} C_VEL
LIN {X 0,Y 493.46,Z 635.51,A -85,B 0,C 180,E1 23241.833,E2 23241.833} C_VEL
LIN {X 0,Y 492.401,Z 652.08,A -85,B 0,C 180,E1 23240.504,E2 23240.504} C_VEL
LIN {X 0,Y 491.319,Z 667.984,A -85,B 0,C 180,E1 23238.94,E2 23238.94} C_VEL
LIN {X 0,Y 490.392,Z 681.604,A -85,B 0,C 180,E1 23237.318,E2 23237.318} C_VEL
LIN {X 0,Y 489.587,Z 694.29,A -85,B 0,C 180,E1 23235.517,E2 23235.517} C_VEL
LIN {X 0,Y 488.956,Z 705.523,A -85,B 0,C 180,E1 23233.601,E2 23233.601} C_VEL
LIN {X 0,Y 488.485,Z 715.203,A -85,B 0,C 180,E1 23231.571,E2 23231.571} C_VEL
LIN {X 0,Y 488.193,Z 722.984,A -85,B 0,C 180,E1 23229.549,E2 23229.549} C_VEL
LIN {X 0,Y 488.016,Z 729.439,A -85,B 0,C 180,E1 23227.414,E2 23227.414} C_VEL
LIN {X 0,Y 487.942,Z 734.377,A -85,B 0,C 180,E1 23225.173,E2 23225.173} C_VEL
LIN {X 0,Y 487.914,Z 737.456,A -85,B 0,C 180,E1 23222.936,E2 23222.936} C_VEL
LIN {X 0,Y 487.915,Z 738.848,A -85,B 0,C 180,E1 23220.704,E2 23220.704} C_VEL
LIN {X 0,Y 487.91,Z 738.609,A -85,B 0,C 180,E1 23218.473,E2 23218.473} C_VEL
LIN {X 0,Y 487.913,Z 736.653,A -85,B 0,C 180,E1 23216.24,E2 23216.24} C_VEL
LIN {X 0,Y 487.951,Z 733.154,A -85,B 0,C 180,E1 23214.119,E2 23214.119} C_VEL
LIN {X 0,Y 488.057,Z 727.733,A -85,B 0,C 180,E1 23211.873,E2 23211.873} C_VEL
LIN {X 0,Y 488.263,Z 720.817,A -85,B 0,C 180,E1 23209.737,E2 23209.737} C_VEL
LIN {X 0,Y 488.632,Z 711.886,A -85,B 0,C 180,E1 23207.592,E2 23207.592} C_VEL
LIN {X 0,Y 489.135,Z 702.017,A -85,B 0,C 180,E1 23205.679,E2 23205.679} C_VEL
LIN {X 0,Y 489.844,Z 690.087,A -85,B 0,C 180,E1 23203.761,E2 23203.761} C_VEL
LIN {X 0,Y 490.706,Z 677.104,A -85,B 0,C 180,E1 23202.019,E2 23202.019} C_VEL
LIN {X 0,Y 491.645,Z 663.277,A -85,B 0,C 180,E1 23200.472,E2 23200.472} C_VEL
LIN {X 0,Y 492.729,Z 647.16,A -85,B 0,C 180,E1 23198.98,E2 23198.98} C_VEL
LIN {X 0,Y 493.811,Z 630.211,A -85,B 0,C 180,E1 23197.694,E2 23197.694} C_VEL
LIN {X 0,Y 494.783,Z 613.369,A -85,B 0,C 180,E1 23196.666,E2 23196.666} C_VEL
LIN {X 0,Y 495.718,Z 594.597,A -85,B 0,C 180,E1 23195.766,E2 23195.766} C_VEL
LIN {X 0,Y 496.477,Z 575.311,A -85,B 0,C 180,E1 23195.08,E2 23195.08} C_VEL
LIN {X 0,Y 497.033,Z 555.361,A -85,B 0,C 180,E1 23194.608,E2 23194.608} C_VEL
LIN {X 0,Y 499.659,Z 359.486,A -85,B 0,C 180,E1 23191.54,E2 23191.54} C_VEL
LIN {X 0,Y 496.729,Z 341.654,A -85,B 0,C 180,E1 23191.013,E2 23191.013} C_VEL
LIN {X 0,Y 496.832,Z 338.92,A -85,B 0,C 180,E1 23190.787,E2 23190.787} C_VEL
LIN {X 0,Y 496.258,Z 333.047,A -85,B 0,C 180,E1 23190.205,E2 23190.205} C_VEL
LIN {X 0,Y 491.542,Z 318.436,A -85,B 0,C 180,E1 23188.498,E2 23188.498} C_VEL
LIN {X 0,Y 491.19,Z 313.389,A -85,B 0,C 180,E1 23187.99,E2 23187.99} C_VEL
LIN {X 0,Y 491.549,Z 306.605,A -85,B 0,C 180,E1 23187.365,E2 23187.365} C_VEL
LIN {X 0,Y 484.858,Z 287.583,A -85,B 0,C 180,E1 23184.954,E2 23184.954} C_VEL
LIN {X 0,Y 480.892,Z 276.792,A -85,B 0,C 180,E1 23183.461,E2 23183.461} C_VEL
LIN {X 0,Y 480.861,Z 276.584,A -85,B 0,C 180,E1 23179.865,E2 23179.865} C_VEL
LIN {X 0,Y 480.883,Z 276.581,A -85,B 0,C 180,E1 23176.345,E2 23176.345} C_VEL
LIN {X 0,Y 480.889,Z 276.582,A -85,B 0,C 180,E1 23172.78,E2 23172.78} C_VEL
LIN {X 0,Y 480.885,Z 276.586,A -85,B 0,C 180,E1 23169.145,E2 23169.145} C_VEL
LIN {X 0,Y 480.887,Z 276.586,A -85,B 0,C 180,E1 23165.605,E2 23165.605} C_VEL
LIN {X 0,Y 480.89,Z 276.583,A -85,B 0,C 180,E1 23161.971,E2 23161.971} C_VEL
LIN {X 0,Y 480.888,Z 276.575,A -85,B 0,C 180,E1 23158.417,E2 23158.417} C_VEL
LIN {X 0,Y 480.859,Z 276.576,A -85,B 0,C 180,E1 23154.837,E2 23154.837} C_VEL
LIN {X 0,Y 480.852,Z 276.58,A -85,B 0,C 180,E1 23151.212,E2 23151.212} C_VEL
LIN {X 0,Y 480.869,Z 276.581,A -85,B 0,C 180,E1 23147.673,E2 23147.673} C_VEL
LIN {X 0,Y 480.891,Z 276.549,A -85,B 0,C 180,E1 23144.08,E2 23144.08} C_VEL
LIN {X 0,Y 480.918,Z 276.848,A -85,B 0,C 180,E1 23142.094,E2 23142.094} C_VEL
LIN {X 0,Y 488.444,Z 299.45,A -85,B 0,C 180,E1 23139.605,E2 23139.605} C_VEL
LIN {X 0,Y 489.329,Z 303.139,A -85,B 0,C 180,E1 23139.231,E2 23139.231} C_VEL
LIN {X 0,Y 488.397,Z 344.101,A -85,B 0,C 180,E1 23135.817,E2 23135.817} C_VEL
LIN {X 0,Y 487.266,Z 385.057,A -85,B 0,C 180,E1 23132.412,E2 23132.412} C_VEL
LIN {X 0,Y 485.959,Z 428.308,A -85,B 0,C 180,E1 23128.822,E2 23128.822} C_VEL
LIN {X 0,Y 484.782,Z 468.905,A -85,B 0,C 180,E1 23125.447,E2 23125.447} C_VEL
LIN {X 0,Y 484.71,Z 475.67,A -85,B 0,C 180,E1 23124.938,E2 23124.938} C_VEL
LIN {X 0,Y 485.868,Z 487.443,A -85,B 0,C 180,E1 23124.705,E2 23124.705} C_VEL
LIN {X 0,Y 484.673,Z 618.138,A -85,B 0,C 180,E1 23122.709,E2 23122.709} C_VEL
LIN {X 0,Y 484.347,Z 634.096,A -85,B 0,C 180,E1 23122.248,E2 23122.248} C_VEL
LIN {X 0,Y 483.857,Z 649.838,A -85,B 0,C 180,E1 23121.565,E2 23121.565} C_VEL
LIN {X 0,Y 483.274,Z 664.307,A -85,B 0,C 180,E1 23120.712,E2 23120.712} C_VEL
LIN {X 0,Y 482.589,Z 678.583,A -85,B 0,C 180,E1 23119.617,E2 23119.617} C_VEL
LIN {X 0,Y 481.968,Z 691.229,A -85,B 0,C 180,E1 23118.393,E2 23118.393} C_VEL
LIN {X 0,Y 481.338,Z 703.356,A -85,B 0,C 180,E1 23116.915,E2 23116.915} C_VEL
LIN {X 0,Y 480.861,Z 713.157,A -85,B 0,C 180,E1 23115.43,E2 23115.43} C_VEL
LIN {X 0,Y 480.457,Z 722.223,A -85,B 0,C 180,E1 23113.685,E2 23113.685} C_VEL
LIN {X 0,Y 480.208,Z 729.304,A -85,B 0,C 180,E1 23111.928,E2 23111.928} C_VEL
LIN {X 0,Y 480.056,Z 734.869,A -85,B 0,C 180,E1 23110.029,E2 23110.029} C_VEL
LIN {X 0,Y 479.989,Z 738.645,A -85,B 0,C 180,E1 23108.109,E2 23108.109} C_VEL
LIN {X 0,Y 479.965,Z 740.614,A -85,B 0,C 180,E1 23106.139,E2 23106.139} C_VEL
LIN {X 0,Y 479.965,Z 740.831,A -85,B 0,C 180,E1 23104.151,E2 23104.151} C_VEL
LIN {X 0,Y 479.982,Z 739.18,A -85,B 0,C 180,E1 23102.187,E2 23102.187} C_VEL
LIN {X 0,Y 480.042,Z 735.885,A -85,B 0,C 180,E1 23100.285,E2 23100.285} C_VEL
LIN {X 0,Y 480.169,Z 730.727,A -85,B 0,C 180,E1 23098.394,E2 23098.394} C_VEL
LIN {X 0,Y 480.415,Z 723.707,A -85,B 0,C 180,E1 23096.53,E2 23096.53} C_VEL
LIN {X 0,Y 480.778,Z 715.173,A -85,B 0,C 180,E1 23094.817,E2 23094.817} C_VEL
LIN {X 0,Y 481.28,Z 704.964,A -85,B 0,C 180,E1 23093.196,E2 23093.196} C_VEL
LIN {X 0,Y 481.872,Z 693.376,A -85,B 0,C 180,E1 23091.742,E2 23091.742} C_VEL
LIN {X 0,Y 482.539,Z 680.323,A -85,B 0,C 180,E1 23090.428,E2 23090.428} C_VEL
LIN {X 0,Y 483.198,Z 666.3,A -85,B 0,C 180,E1 23089.324,E2 23089.324} C_VEL
LIN {X 0,Y 483.819,Z 651.659,A -85,B 0,C 180,E1 23088.428,E2 23088.428} C_VEL
LIN {X 0,Y 484.321,Z 635.548,A -85,B 0,C 180,E1 23087.71,E2 23087.71} C_VEL
LIN {X 0,Y 484.657,Z 619.372,A -85,B 0,C 180,E1 23087.222,E2 23087.222} C_VEL
LIN {X 0,Y 485.06,Z 573.604,A -85,B 0,C 180,E1 23086.498,E2 23086.498} C_VEL
LIN {X 0,Y 485.702,Z 483.779,A -85,B 0,C 180,E1 23085.133,E2 23085.133} C_VEL
LIN {X 0,Y 484.654,Z 474.864,A -85,B 0,C 180,E1 23084.917,E2 23084.917} C_VEL
LIN {X 0,Y 485.874,Z 430.646,A -85,B 0,C 180,E1 23081.274,E2 23081.274} C_VEL
LIN {X 0,Y 487.07,Z 390.003,A -85,B 0,C 180,E1 23077.939,E2 23077.939} C_VEL
LIN {X 0,Y 487.969,Z 349.682,A -85,B 0,C 180,E1 23074.654,E2 23074.654} C_VEL
LIN {X 0,Y 488.646,Z 311.158,A -85,B 0,C 180,E1 23071.521,E2 23071.521} C_VEL
LIN {X 0,Y 488.615,Z 300.388,A -85,B 0,C 180,E1 23070.633,E2 23070.633} C_VEL
LIN {X 0,Y 481.718,Z 279.355,A -85,B 0,C 180,E1 23068.448,E2 23068.448} C_VEL
LIN {X 0,Y 480.89,Z 276.79,A -85,B 0,C 180,E1 23068.119,E2 23068.119} C_VEL
LIN {X 0,Y 480.851,Z 276.59,A -85,B 0,C 180,E1 23064.575,E2 23064.575} C_VEL
LIN {X 0,Y 480.873,Z 276.581,A -85,B 0,C 180,E1 23061.005,E2 23061.005} C_VEL
LIN {X 0,Y 480.895,Z 276.586,A -85,B 0,C 180,E1 23057.389,E2 23057.389} C_VEL
LIN {X 0,Y 480.874,Z 276.588,A -85,B 0,C 180,E1 23053.835,E2 23053.835} C_VEL
LIN {X 0,Y 480.852,Z 276.585,A -85,B 0,C 180,E1 23050.302,E2 23050.302} C_VEL
LIN {X 0,Y 480.861,Z 276.582,A -85,B 0,C 180,E1 23046.687,E2 23046.687} C_VEL
LIN {X 0,Y 480.889,Z 276.583,A -85,B 0,C 180,E1 23043.099,E2 23043.099} C_VEL
LIN {X 0,Y 480.891,Z 276.584,A -85,B 0,C 180,E1 23039.524,E2 23039.524} C_VEL
LIN {X 0,Y 480.859,Z 276.584,A -85,B 0,C 180,E1 23035.946,E2 23035.946} C_VEL
LIN {X 0,Y 480.857,Z 276.583,A -85,B 0,C 180,E1 23032.353,E2 23032.353} C_VEL
LIN {X 0,Y 480.884,Z 276.582,A -85,B 0,C 180,E1 23028.851,E2 23028.851} C_VEL
LIN {X 0,Y 480.896,Z 276.581,A -85,B 0,C 180,E1 23025.189,E2 23025.189} C_VEL
LIN {X 0,Y 480.875,Z 276.586,A -85,B 0,C 180,E1 23021.576,E2 23021.576} C_VEL
LIN {X 0,Y 480.856,Z 276.582,A -85,B 0,C 180,E1 23018.021,E2 23018.021} C_VEL
LIN {X 0,Y 480.874,Z 276.582,A -85,B 0,C 180,E1 23014.47,E2 23014.47} C_VEL
LIN {X 0,Y 480.897,Z 276.579,A -85,B 0,C 180,E1 23010.834,E2 23010.834} C_VEL
LIN {X 0,Y 480.888,Z 276.586,A -85,B 0,C 180,E1 23007.277,E2 23007.277} C_VEL
LIN {X 0,Y 480.864,Z 276.585,A -85,B 0,C 180,E1 23003.659,E2 23003.659} C_VEL
LIN {X 0,Y 480.863,Z 276.584,A -85,B 0,C 180,E1 23000.022,E2 23000.022} C_VEL
LIN {X 0,Y 480.888,Z 276.584,A -85,B 0,C 180,E1 22996.512,E2 22996.512} C_VEL
LIN {X 0,Y 480.893,Z 276.584,A -85,B 0,C 180,E1 22992.832,E2 22992.832} C_VEL
LIN {X 0,Y 480.885,Z 276.658,A -85,B 0,C 180,E1 22989.334,E2 22989.334} C_VEL
LIN {X 0,Y 481.011,Z 277.282,A -85,B 0,C 180,E1 22989.111,E2 22989.111} C_VEL
LIN {X 0,Y 489.24,Z 297.693,A -85,B 0,C 180,E1 22986.566,E2 22986.566} C_VEL
LIN {X 0,Y 493.883,Z 310.615,A -85,B 0,C 180,E1 22985.094,E2 22985.094} C_VEL
LIN {X 0,Y 493.628,Z 317.053,A -85,B 0,C 180,E1 22984.621,E2 22984.621} C_VEL
LIN {X 0,Y 496.497,Z 336.987,A -85,B 0,C 180,E1 22984.03,E2 22984.03} C_VEL
LIN {X 0,Y 493.015,Z 543.06,A -85,B 0,C 180,E1 22980.681,E2 22980.681} C_VEL
LIN {X 0,Y 492.461,Z 578.367,A -85,B 0,C 180,E1 22980.102,E2 22980.102} C_VEL
LIN {X 0,Y 491.654,Z 599.684,A -85,B 0,C 180,E1 22979.538,E2 22979.538} C_VEL
LIN {X 0,Y 490.64,Z 620.714,A -85,B 0,C 180,E1 22978.745,E2 22978.745} C_VEL
LIN {X 0,Y 489.439,Z 640.672,A -85,B 0,C 180,E1 22977.758,E2 22977.758} C_VEL
LIN {X 0,Y 488.164,Z 659.689,A -85,B 0,C 180,E1 22976.584,E2 22976.584} C_VEL
LIN {X 0,Y 486.856,Z 677.606,A -85,B 0,C 180,E1 22975.241,E2 22975.241} C_VEL
LIN {X 0,Y 485.499,Z 695.057,A -85,B 0,C 180,E1 22973.676,E2 22973.676} C_VEL
LIN {X 0,Y 484.298,Z 710.567,A -85,B 0,C 180,E1 22972.031,E2 22972.031} C_VEL
LIN {X 0,Y 483.184,Z 725.151,A -85,B 0,C 180,E1 22970.215,E2 22970.215} C_VEL
LIN {X 0,Y 482.158,Z 739.298,A -85,B 0,C 180,E1 22968.121,E2 22968.121} C_VEL
LIN {X 0,Y 481.323,Z 751.868,A -85,B 0,C 180,E1 22965.889,E2 22965.889} C_VEL
LIN {X 0,Y 480.793,Z 760.85,A -85,B 0,C 180,E1 22963.958,E2 22963.958} C_VEL
LIN {X 0,Y 480.355,Z 769.658,A -85,B 0,C 180,E1 22961.647,E2 22961.647} C_VEL
LIN {X 0,Y 480.097,Z 776.687,A -85,B 0,C 180,E1 22959.347,E2 22959.347} C_VEL
LIN {X 0,Y 479.971,Z 782.262,A -85,B 0,C 180,E1 22956.938,E2 22956.938} C_VEL
LIN {X 0,Y 479.919,Z 786.088,A -85,B 0,C 180,E1 22954.539,E2 22954.539} C_VEL
LIN {X 0,Y 479.909,Z 788.304,A -85,B 0,C 180,E1 22952.148,E2 22952.148} C_VEL
LIN {X 0,Y 479.905,Z 788.961,A -85,B 0,C 180,E1 22949.76,E2 22949.76} C_VEL
LIN {X 0,Y 479.909,Z 788.029,A -85,B 0,C 180,E1 22947.372,E2 22947.372} C_VEL
LIN {X 0,Y 479.923,Z 785.444,A -85,B 0,C 180,E1 22944.979,E2 22944.979} C_VEL
LIN {X 0,Y 479.982,Z 781.182,A -85,B 0,C 180,E1 22942.55,E2 22942.55} C_VEL
LIN {X 0,Y 480.145,Z 775.322,A -85,B 0,C 180,E1 22940.167,E2 22940.167} C_VEL
LIN {X 0,Y 480.43,Z 768.003,A -85,B 0,C 180,E1 22937.865,E2 22937.865} C_VEL
LIN {X 0,Y 480.913,Z 758.779,A -85,B 0,C 180,E1 22935.552,E2 22935.552} C_VEL
LIN {X 0,Y 481.481,Z 749.052,A -85,B 0,C 180,E1 22933.594,E2 22933.594} C_VEL
LIN {X 0,Y 482.295,Z 736.669,A -85,B 0,C 180,E1 22931.506,E2 22931.506} C_VEL
LIN {X 0,Y 483.24,Z 723.261,A -85,B 0,C 180,E1 22929.601,E2 22929.601} C_VEL
LIN {X 0,Y 484.338,Z 708.311,A -85,B 0,C 180,E1 22927.803,E2 22927.803} C_VEL
LIN {X 0,Y 485.572,Z 691.104,A -85,B 0,C 180,E1 22926.067,E2 22926.067} C_VEL
LIN {X 0,Y 486.801,Z 673.363,A -85,B 0,C 180,E1 22924.578,E2 22924.578} C_VEL
LIN {X 0,Y 487.986,Z 654.951,A -85,B 0,C 180,E1 22923.296,E2 22923.296} C_VEL
LIN {X 0,Y 489.066,Z 636.002,A -85,B 0,C 180,E1 22922.216,E2 22922.216} C_VEL
LIN {X 0,Y 490.074,Z 615.351,A -85,B 0,C 180,E1 22921.283,E2 22921.283} C_VEL
LIN {X 0,Y 490.923,Z 594.202,A -85,B 0,C 180,E1 22920.569,E2 22920.569} C_VEL
LIN {X 0,Y 491.499,Z 573.212,A -85,B 0,C 180,E1 22920.081,E2 22920.081} C_VEL
LIN {X 0,Y 493.426,Z 427.106,A -85,B 0,C 180,E1 22917.78,E2 22917.78} C_VEL
LIN {X 0,Y 495.194,Z 334.57,A -85,B 0,C 180,E1 22916.154,E2 22916.154} C_VEL
LIN {X 0,Y 493.038,Z 318.591,A -85,B 0,C 180,E1 22915.626,E2 22915.626} C_VEL
LIN {X 0,Y 493.51,Z 309.486,A -85,B 0,C 180,E1 22914.872,E2 22914.872} C_VEL
LIN {X 0,Y 488.887,Z 295.609,A -85,B 0,C 180,E1 22913.097,E2 22913.097} C_VEL
LIN {X 0,Y 485.637,Z 287.551,A -85,B 0,C 180,E1 22911.854,E2 22911.854} C_VEL
LIN {X 0,Y 482.851,Z 280.995,A -85,B 0,C 180,E1 22910.679,E2 22910.679} C_VEL
LIN {X 0,Y 481.021,Z 277.436,A -85,B 0,C 180,E1 22909.88,E2 22909.88} C_VEL
LIN {X 0,Y 480.9,Z 276.647,A -85,B 0,C 180,E1 22909.549,E2 22909.549} C_VEL
LIN {X 0,Y 480.86,Z 276.588,A -85,B 0,C 180,E1 22906.008,E2 22906.008} C_VEL
LIN {X 0,Y 480.854,Z 276.59,A -85,B 0,C 180,E1 22902.353,E2 22902.353} C_VEL
LIN {X 0,Y 480.885,Z 276.587,A -85,B 0,C 180,E1 22898.896,E2 22898.896} C_VEL
LIN {X 0,Y 480.911,Z 276.996,A -85,B 0,C 180,E1 22898.224,E2 22898.224} C_VEL
LIN {X 0,Y 482.518,Z 280.522,A -85,B 0,C 180,E1 22897.383,E2 22897.383} C_VEL
LIN {X 0,Y 486.264,Z 289.034,A -85,B 0,C 180,E1 22895.687,E2 22895.687} C_VEL
LIN {X 0,Y 490.455,Z 300.635,A -85,B 0,C 180,E1 22893.817,E2 22893.817} C_VEL
LIN {X 0,Y 492.865,Z 308.324,A -85,B 0,C 180,E1 22892.727,E2 22892.727} C_VEL
LIN {X 0,Y 490.407,Z 340.423,A -85,B 0,C 180,E1 22889.709,E2 22889.709} C_VEL
LIN {X 0,Y 493.622,Z 361.673,A -85,B 0,C 180,E1 22888.962,E2 22888.962} C_VEL
LIN {X 0,Y 490.92,Z 469.402,A -85,B 0,C 180,E1 22887.045,E2 22887.045} C_VEL
LIN {X 0,Y 489.387,Z 562.174,A -85,B 0,C 180,E1 22885.496,E2 22885.496} C_VEL
LIN {X 0,Y 488.743,Z 581.455,A -85,B 0,C 180,E1 22884.965,E2 22884.965} C_VEL
LIN {X 0,Y 487.918,Z 600.195,A -85,B 0,C 180,E1 22884.228,E2 22884.228} C_VEL
LIN {X 0,Y 486.949,Z 618.418,A -85,B 0,C 180,E1 22883.282,E2 22883.282} C_VEL
LIN {X 0,Y 485.86,Z 636.052,A -85,B 0,C 180,E1 22882.123,E2 22882.123} C_VEL
LIN {X 0,Y 484.742,Z 652.559,A -85,B 0,C 180,E1 22880.779,E2 22880.779} C_VEL
LIN {X 0,Y 483.633,Z 667.932,A -85,B 0,C 180,E1 22879.253,E2 22879.253} C_VEL
LIN {X 0,Y 482.641,Z 681.672,A -85,B 0,C 180,E1 22877.605,E2 22877.605} C_VEL
LIN {X 0,Y 481.764,Z 694.357,A -85,B 0,C 180,E1 22875.776,E2 22875.776} C_VEL
LIN {X 0,Y 481.064,Z 705.528,A -85,B 0,C 180,E1 22873.828,E2 22873.828} C_VEL
LIN {X 0,Y 480.549,Z 715.203,A -85,B 0,C 180,E1 22871.765,E2 22871.765} C_VEL
LIN {X 0,Y 480.226,Z 722.986,A -85,B 0,C 180,E1 22869.709,E2 22869.709} C_VEL
LIN {X 0,Y 480.024,Z 729.574,A -85,B 0,C 180,E1 22867.482,E2 22867.482} C_VEL
LIN {X 0,Y 479.944,Z 734.41,A -85,B 0,C 180,E1 22865.242,E2 22865.242} C_VEL
LIN {X 0,Y 479.914,Z 737.453,A -85,B 0,C 180,E1 22862.985,E2 22862.985} C_VEL
LIN {X 0,Y 479.915,Z 738.847,A -85,B 0,C 180,E1 22860.716,E2 22860.716} C_VEL
LIN {X 0,Y 479.912,Z 738.677,A -85,B 0,C 180,E1 22858.567,E2 22858.567} C_VEL
LIN {X 0,Y 479.914,Z 736.777,A -85,B 0,C 180,E1 22856.296,E2 22856.296} C_VEL
LIN {X 0,Y 479.952,Z 733.384,A -85,B 0,C 180,E1 22854.141,E2 22854.141} C_VEL
LIN {X 0,Y 480.054,Z 728.422,A -85,B 0,C 180,E1 22851.978,E2 22851.978} C_VEL
LIN {X 0,Y 480.269,Z 721.665,A -85,B 0,C 180,E1 22849.807,E2 22849.807} C_VEL
LIN {X 0,Y 480.626,Z 713.468,A -85,B 0,C 180,E1 22847.749,E2 22847.749} C_VEL
LIN {X 0,Y 481.227,Z 702.728,A -85,B 0,C 180,E1 22845.562,E2 22845.562} C_VEL
LIN {X 0,Y 482.046,Z 690.126,A -85,B 0,C 180,E1 22843.491,E2 22843.491} C_VEL
LIN {X 0,Y 482.943,Z 677.594,A -85,B 0,C 180,E1 22841.782,E2 22841.782} C_VEL
LIN {X 0,Y 483.961,Z 663.643,A -85,B 0,C 180,E1 22840.194,E2 22840.194} C_VEL
LIN {X 0,Y 485.114,Z 647.635,A -85,B 0,C 180,E1 22838.688,E2 22838.688} C_VEL
LIN {X 0,Y 486.263,Z 630.749,A -85,B 0,C 180,E1 22837.386,E2 22837.386} C_VEL
LIN {X 0,Y 487.349,Z 612.991,A -85,B 0,C 180,E1 22836.289,E2 22836.289} C_VEL
LIN {X 0,Y 488.362,Z 594.03,A -85,B 0,C 180,E1 22835.373,E2 22835.373} C_VEL
LIN {X 0,Y 489.175,Z 574.432,A -85,B 0,C 180,E1 22834.678,E2 22834.678} C_VEL
LIN {X 0,Y 489.759,Z 554.493,A -85,B 0,C 180,E1 22834.209,E2 22834.209} C_VEL
LIN {X 0,Y 492.703,Z 360.753,A -85,B 0,C 180,E1 22831.099,E2 22831.099} C_VEL
LIN {X 0,Y 489.554,Z 341.423,A -85,B 0,C 180,E1 22830.513,E2 22830.513} C_VEL
LIN {X 0,Y 491.19,Z 313.389,A -85,B 0,C 180,E1 22827.99,E2 22827.99} C_VEL
LIN {X 0,Y 490.515,Z 310.28,A -85,B 0,C 180,E1 22827.641,E2 22827.641} C_VEL
LIN {X 0,Y 487.47,Z 306.792,A -85,B 0,C 180,E1 22827.068,E2 22827.068} C_VEL
LIN {X 0,Y 482.264,Z 302.171,A -85,B 0,C 180,E1 22826.196,E2 22826.196} C_VEL
LIN {X 0,Y 481.268,Z 300.303,A -85,B 0,C 180,E1 22825.928,E2 22825.928} C_VEL
LIN {X 0,Y 473.968,Z 280.663,A -85,B 0,C 180,E1 22823.287,E2 22823.287} C_VEL
LIN {X 0,Y 472.982,Z 277.764,A -85,B 0,C 180,E1 22822.842,E2 22822.842} C_VEL
LIN {X 0,Y 472.955,Z 277.574,A -85,B 0,C 180,E1 22819.187,E2 22819.187} C_VEL
LIN {X 0,Y 472.937,Z 277.569,A -85,B 0,C 180,E1 22815.59,E2 22815.59} C_VEL
LIN {X 0,Y 472.937,Z 277.574,A -85,B 0,C 180,E1 22811.91,E2 22811.91} C_VEL
LIN {X 0,Y 472.95,Z 277.57,A -85,B 0,C 180,E1 22808.275,E2 22808.275} C_VEL
LIN {X 0,Y 472.943,Z 277.57,A -85,B 0,C 180,E1 22804.661,E2 22804.661} C_VEL
LIN {X 0,Y 472.932,Z 277.57,A -85,B 0,C 180,E1 22801.056,E2 22801.056} C_VEL
LIN {X 0,Y 472.94,Z 277.577,A -85,B 0,C 180,E1 22797.445,E2 22797.445} C_VEL
LIN {X 0,Y 472.954,Z 277.568,A -85,B 0,C 180,E1 22793.816,E2 22793.816} C_VEL
LIN {X 0,Y 472.952,Z 277.57,A -85,B 0,C 180,E1 22790.158,E2 22790.158} C_VEL
LIN {X 0,Y 472.916,Z 277.578,A -85,B 0,C 180,E1 22786.585,E2 22786.585} C_VEL
LIN {X 0,Y 472.888,Z 277.551,A -85,B 0,C 180,E1 22783.077,E2 22783.077} C_VEL
LIN {X 0,Y 472.949,Z 277.865,A -85,B 0,C 180,E1 22782.578,E2 22782.578} C_VEL
LIN {X 0,Y 480.124,Z 299.048,A -85,B 0,C 180,E1 22780.197,E2 22780.197} C_VEL
LIN {X 0,Y 482.022,Z 305.695,A -85,B 0,C 180,E1 22779.493,E2 22779.493} C_VEL
LIN {X 0,Y 480.988,Z 346.959,A -85,B 0,C 180,E1 22776.027,E2 22776.027} C_VEL
LIN {X 0,Y 479.767,Z 388.214,A -85,B 0,C 180,E1 22772.569,E2 22772.569} C_VEL
LIN {X 0,Y 478.381,Z 431.042,A -85,B 0,C 180,E1 22768.983,E2 22768.983} C_VEL
LIN {X 0,Y 477.128,Z 471.961,A -85,B 0,C 180,E1 22765.554,E2 22765.554} C_VEL
LIN {X 0,Y 477.145,Z 476.184,A -85,B 0,C 180,E1 22765.261,E2 22765.261} C_VEL
LIN {X 0,Y 478.337,Z 488.23,A -85,B 0,C 180,E1 22765.017,E2 22765.017} C_VEL
LIN {X 0,Y 477.055,Z 618.508,A -85,B 0,C 180,E1 22762.996,E2 22762.996} C_VEL
LIN {X 0,Y 476.711,Z 634.427,A -85,B 0,C 180,E1 22762.53,E2 22762.53} C_VEL
LIN {X 0,Y 476.189,Z 650.185,A -85,B 0,C 180,E1 22761.836,E2 22761.836} C_VEL
LIN {X 0,Y 475.581,Z 664.381,A -85,B 0,C 180,E1 22760.99,E2 22760.99} C_VEL
LIN {X 0,Y 474.845,Z 678.749,A -85,B 0,C 180,E1 22759.875,E2 22759.875} C_VEL
LIN {X 0,Y 474.191,Z 691.16,A -85,B 0,C 180,E1 22758.664,E2 22758.664} C_VEL
LIN {X 0,Y 473.516,Z 703.151,A -85,B 0,C 180,E1 22757.192,E2 22757.192} C_VEL
LIN {X 0,Y 472.991,Z 713.077,A -85,B 0,C 180,E1 22755.682,E2 22755.682} C_VEL
LIN {X 0,Y 472.568,Z 721.663,A -85,B 0,C 180,E1 22754.036,E2 22754.036} C_VEL
LIN {X 0,Y 472.273,Z 728.948,A -85,B 0,C 180,E1 22752.252,E2 22752.252} C_VEL
LIN {X 0,Y 472.1,Z 734.434,A -85,B 0,C 180,E1 22750.452,E2 22750.452} C_VEL
LIN {X 0,Y 472.007,Z 738.604,A -85,B 0,C 180,E1 22748.427,E2 22748.427} C_VEL
LIN {X 0,Y 471.978,Z 740.795,A -85,B 0,C 180,E1 22746.532,E2 22746.532} C_VEL
LIN {X 0,Y 471.972,Z 741.29,A -85,B 0,C 180,E1 22744.486,E2 22744.486} C_VEL
LIN {X 0,Y 471.99,Z 740.026,A -85,B 0,C 180,E1 22742.498,E2 22742.498} C_VEL
LIN {X 0,Y 472.047,Z 736.922,A -85,B 0,C 180,E1 22740.524,E2 22740.524} C_VEL
LIN {X 0,Y 472.178,Z 732.074,A -85,B 0,C 180,E1 22738.581,E2 22738.581} C_VEL
LIN {X 0,Y 472.419,Z 725.464,A -85,B 0,C 180,E1 22736.722,E2 22736.722} C_VEL
LIN {X 0,Y 472.807,Z 717.11,A -85,B 0,C 180,E1 22734.926,E2 22734.926} C_VEL
LIN {X 0,Y 473.315,Z 707.291,A -85,B 0,C 180,E1 22733.288,E2 22733.288} C_VEL
LIN {X 0,Y 473.945,Z 696.083,A -85,B 0,C 180,E1 22731.787,E2 22731.787} C_VEL
LIN {X 0,Y 474.629,Z 683.459,A -85,B 0,C 180,E1 22730.447,E2 22730.447} C_VEL
LIN {X 0,Y 475.342,Z 670.013,A -85,B 0,C 180,E1 22729.305,E2 22729.305} C_VEL
LIN {X 0,Y 476.011,Z 655.204,A -85,B 0,C 180,E1 22728.335,E2 22728.335} C_VEL
LIN {X 0,Y 476.565,Z 640.458,A -85,B 0,C 180,E1 22727.606,E2 22727.606} C_VEL
LIN {X 0,Y 476.958,Z 624.513,A -85,B 0,C 180,E1 22727.057,E2 22727.057} C_VEL
LIN {X 0,Y 477.191,Z 606.756,A -85,B 0,C 180,E1 22726.697,E2 22726.697} C_VEL
LIN {X 0,Y 478.186,Z 484.616,A -85,B 0,C 180,E1 22724.815,E2 22724.815} C_VEL
LIN {X 0,Y 477.083,Z 475.353,A -85,B 0,C 180,E1 22724.595,E2 22724.595} C_VEL
LIN {X 0,Y 478.366,Z 431.489,A -85,B 0,C 180,E1 22720.95,E2 22720.95} C_VEL
LIN {X 0,Y 479.648,Z 390.654,A -85,B 0,C 180,E1 22717.571,E2 22717.571} C_VEL
LIN {X 0,Y 480.647,Z 348.534,A -85,B 0,C 180,E1 22714.116,E2 22714.116} C_VEL
LIN {X 0,Y 481.427,Z 308.035,A -85,B 0,C 180,E1 22710.794,E2 22710.794} C_VEL
LIN {X 0,Y 481.348,Z 303.12,A -85,B 0,C 180,E1 22710.385,E2 22710.385} C_VEL
LIN {X 0,Y 474.821,Z 283.199,A -85,B 0,C 180,E1 22708.282,E2 22708.282} C_VEL
LIN {X 0,Y 473,Z 277.889,A -85,B 0,C 180,E1 22707.665,E2 22707.665} C_VEL
LIN {X 0,Y 472.915,Z 277.578,A -85,B 0,C 180,E1 22706.766,E2 22706.766} C_VEL
LIN {X 0,Y 472.943,Z 277.572,A -85,B 0,C 180,E1 22703.156,E2 22703.156} C_VEL
LIN {X 0,Y 472.954,Z 277.571,A -85,B 0,C 180,E1 22699.514,E2 22699.514} C_VEL
LIN {X 0,Y 472.933,Z 277.572,A -85,B 0,C 180,E1 22695.865,E2 22695.865} C_VEL
LIN {X 0,Y 472.912,Z 277.575,A -85,B 0,C 180,E1 22692.33,E2 22692.33} C_VEL
LIN {X 0,Y 472.926,Z 277.571,A -85,B 0,C 180,E1 22688.756,E2 22688.756} C_VEL
LIN {X 0,Y 472.953,Z 277.572,A -85,B 0,C 180,E1 22685.216,E2 22685.216} C_VEL
LIN {X 0,Y 472.947,Z 277.573,A -85,B 0,C 180,E1 22681.575,E2 22681.575} C_VEL
LIN {X 0,Y 472.917,Z 277.573,A -85,B 0,C 180,E1 22678.062,E2 22678.062} C_VEL
LIN {X 0,Y 472.919,Z 277.573,A -85,B 0,C 180,E1 22674.419,E2 22674.419} C_VEL
LIN {X 0,Y 472.947,Z 277.567,A -85,B 0,C 180,E1 22670.877,E2 22670.877} C_VEL
LIN {X 0,Y 472.955,Z 277.57,A -85,B 0,C 180,E1 22667.175,E2 22667.175} C_VEL
LIN {X 0,Y 472.939,Z 277.572,A -85,B 0,C 180,E1 22663.543,E2 22663.543} C_VEL
LIN {X 0,Y 472.919,Z 277.573,A -85,B 0,C 180,E1 22659.971,E2 22659.971} C_VEL
LIN {X 0,Y 472.924,Z 277.573,A -85,B 0,C 180,E1 22656.265,E2 22656.265} C_VEL
LIN {X 0,Y 472.947,Z 277.569,A -85,B 0,C 180,E1 22652.609,E2 22652.609} C_VEL
LIN {X 0,Y 472.956,Z 277.571,A -85,B 0,C 180,E1 22648.947,E2 22648.947} C_VEL
LIN {X 0,Y 472.944,Z 277.574,A -85,B 0,C 180,E1 22645.321,E2 22645.321} C_VEL
LIN {X 0,Y 472.924,Z 277.573,A -85,B 0,C 180,E1 22641.724,E2 22641.724} C_VEL
LIN {X 0,Y 472.927,Z 277.574,A -85,B 0,C 180,E1 22638.081,E2 22638.081} C_VEL
LIN {X 0,Y 472.951,Z 277.572,A -85,B 0,C 180,E1 22634.566,E2 22634.566} C_VEL
LIN {X 0,Y 472.958,Z 277.574,A -85,B 0,C 180,E1 22630.944,E2 22630.944} C_VEL
LIN {X 0,Y 472.976,Z 277.929,A -85,B 0,C 180,E1 22629.81,E2 22629.81} C_VEL
LIN {X 0,Y 482.114,Z 300.518,A -85,B 0,C 180,E1 22626.919,E2 22626.919} C_VEL
LIN {X 0,Y 486.799,Z 313.699,A -85,B 0,C 180,E1 22625.393,E2 22625.393} C_VEL
LIN {X 0,Y 486.741,Z 317.483,A -85,B 0,C 180,E1 22625.135,E2 22625.135} C_VEL
LIN {X 0,Y 489.712,Z 338.32,A -85,B 0,C 180,E1 22624.508,E2 22624.508} C_VEL
LIN {X 0,Y 485.818,Z 547.216,A -85,B 0,C 180,E1 22621.041,E2 22621.041} C_VEL
LIN {X 0,Y 485.253,Z 578.797,A -85,B 0,C 180,E1 22620.506,E2 22620.506} C_VEL
LIN {X 0,Y 484.4,Z 599.834,A -85,B 0,C 180,E1 22619.937,E2 22619.937} C_VEL
LIN {X 0,Y 483.303,Z 621.042,A -85,B 0,C 180,E1 22619.121,E2 22619.121} C_VEL
LIN {X 0,Y 481.99,Z 641.435,A -85,B 0,C 180,E1 22618.091,E2 22618.091} C_VEL
LIN {X 0,Y 480.635,Z 660.241,A -85,B 0,C 180,E1 22616.9,E2 22616.9} C_VEL
LIN {X 0,Y 479.226,Z 678.232,A -85,B 0,C 180,E1 22615.519,E2 22615.519} C_VEL
LIN {X 0,Y 477.805,Z 695.344,A -85,B 0,C 180,E1 22613.95,E2 22613.95} C_VEL
LIN {X 0,Y 476.431,Z 711.863,A -85,B 0,C 180,E1 22612.147,E2 22612.147} C_VEL
LIN {X 0,Y 475.271,Z 726.138,A -85,B 0,C 180,E1 22610.31,E2 22610.31} C_VEL
LIN {X 0,Y 474.26,Z 739.363,A -85,B 0,C 180,E1 22608.307,E2 22608.307} C_VEL
LIN {X 0,Y 473.384,Z 751.826,A -85,B 0,C 180,E1 22606.049,E2 22606.049} C_VEL
LIN {X 0,Y 472.771,Z 761.962,A -85,B 0,C 180,E1 22603.825,E2 22603.825} C_VEL
LIN {X 0,Y 472.355,Z 770.304,A -85,B 0,C 180,E1 22601.599,E2 22601.599} C_VEL
LIN {X 0,Y 472.097,Z 777.293,A -85,B 0,C 180,E1 22599.261,E2 22599.261} C_VEL
LIN {X 0,Y 471.974,Z 782.512,A -85,B 0,C 180,E1 22596.934,E2 22596.934} C_VEL
LIN {X 0,Y 471.919,Z 786.247,A -85,B 0,C 180,E1 22594.495,E2 22594.495} C_VEL
LIN {X 0,Y 471.91,Z 788.371,A -85,B 0,C 180,E1 22592.063,E2 22592.063} C_VEL
LIN {X 0,Y 471.901,Z 788.916,A -85,B 0,C 180,E1 22589.513,E2 22589.513} C_VEL
LIN {X 0,Y 471.909,Z 787.843,A -85,B 0,C 180,E1 22587.084,E2 22587.084} C_VEL
LIN {X 0,Y 471.924,Z 785.124,A -85,B 0,C 180,E1 22584.65,E2 22584.65} C_VEL
LIN {X 0,Y 472.014,Z 780.732,A -85,B 0,C 180,E1 22582.207,E2 22582.207} C_VEL
LIN {X 0,Y 472.183,Z 774.94,A -85,B 0,C 180,E1 22579.876,E2 22579.876} C_VEL
LIN {X 0,Y 472.469,Z 767.71,A -85,B 0,C 180,E1 22577.657,E2 22577.657} C_VEL
LIN {X 0,Y 472.982,Z 758.094,A -85,B 0,C 180,E1 22575.304,E2 22575.304} C_VEL
LIN {X 0,Y 473.671,Z 746.862,A -85,B 0,C 180,E1 22573.063,E2 22573.063} C_VEL
LIN {X 0,Y 474.568,Z 734.047,A -85,B 0,C 180,E1 22570.938,E2 22570.938} C_VEL
LIN {X 0,Y 475.639,Z 719.598,A -85,B 0,C 180,E1 22568.932,E2 22568.932} C_VEL
LIN {X 0,Y 476.834,Z 703.931,A -85,B 0,C 180,E1 22567.103,E2 22567.103} C_VEL
LIN {X 0,Y 478.149,Z 686.621,A -85,B 0,C 180,E1 22565.408,E2 22565.408} C_VEL
LIN {X 0,Y 479.426,Z 668.869,A -85,B 0,C 180,E1 22563.959,E2 22563.959} C_VEL
LIN {X 0,Y 480.65,Z 650.205,A -85,B 0,C 180,E1 22562.696,E2 22562.696} C_VEL
LIN {X 0,Y 481.817,Z 630.66,A -85,B 0,C 180,E1 22561.625,E2 22561.625} C_VEL
LIN {X 0,Y 482.816,Z 610.013,A -85,B 0,C 180,E1 22560.742,E2 22560.742} C_VEL
LIN {X 0,Y 483.647,Z 588.937,A -85,B 0,C 180,E1 22560.078,E2 22560.078} C_VEL
LIN {X 0,Y 484.197,Z 567.797,A -85,B 0,C 180,E1 22559.633,E2 22559.633} C_VEL
LIN {X 0,Y 486.013,Z 442.58,A -85,B 0,C 180,E1 22557.612,E2 22557.612} C_VEL
LIN {X 0,Y 488.481,Z 339.694,A -85,B 0,C 180,E1 22555.755,E2 22555.755} C_VEL
LIN {X 0,Y 488.291,Z 334.925,A -85,B 0,C 180,E1 22555.638,E2 22555.638} C_VEL
LIN {X 0,Y 486.291,Z 319.701,A -85,B 0,C 180,E1 22555.122,E2 22555.122} C_VEL
LIN {X 0,Y 486.684,Z 312.859,A -85,B 0,C 180,E1 22554.546,E2 22554.546} C_VEL
LIN {X 0,Y 482.508,Z 299.812,A -85,B 0,C 180,E1 22552.812,E2 22552.812} C_VEL
LIN {X 0,Y 478.669,Z 289.95,A -85,B 0,C 180,E1 22551.181,E2 22551.181} C_VEL
LIN {X 0,Y 476.698,Z 285.829,A -85,B 0,C 180,E1 22550.333,E2 22550.333} C_VEL
LIN {X 0,Y 474.868,Z 281.861,A -85,B 0,C 180,E1 22549.411,E2 22549.411} C_VEL
LIN {X 0,Y 473,Z 278.092,A -85,B 0,C 180,E1 22548.317,E2 22548.317} C_VEL
LIN {X 0,Y 472.946,Z 277.575,A -85,B 0,C 180,E1 22547.591,E2 22547.591} C_VEL
LIN {X 0,Y 472.919,Z 277.579,A -85,B 0,C 180,E1 22544.04,E2 22544.04} C_VEL
LIN {X 0,Y 472.918,Z 277.579,A -85,B 0,C 180,E1 22540.436,E2 22540.436} C_VEL
LIN {X 0,Y 473.012,Z 278.109,A -85,B 0,C 180,E1 22539.749,E2 22539.749} C_VEL
LIN {X 0,Y 474.946,Z 282.011,A -85,B 0,C 180,E1 22538.545,E2 22538.545} C_VEL
LIN {X 0,Y 477.472,Z 287.685,A -85,B 0,C 180,E1 22537.174,E2 22537.174} C_VEL
LIN {X 0,Y 480.774,Z 295.609,A -85,B 0,C 180,E1 22535.593,E2 22535.593} C_VEL
LIN {X 0,Y 484.37,Z 306.095,A -85,B 0,C 180,E1 22533.872,E2 22533.872} C_VEL
LIN {X 0,Y 486.032,Z 311.9,A -85,B 0,C 180,E1 22533.035,E2 22533.035} C_VEL
LIN {X 0,Y 483.594,Z 340.076,A -85,B 0,C 180,E1 22530.326,E2 22530.326} C_VEL
LIN {X 0,Y 487.001,Z 362.667,A -85,B 0,C 180,E1 22529.477,E2 22529.477} C_VEL
LIN {X 0,Y 484.009,Z 460.793,A -85,B 0,C 180,E1 22527.633,E2 22527.633} C_VEL
LIN {X 0,Y 481.994,Z 563.137,A -85,B 0,C 180,E1 22525.846,E2 22525.846} C_VEL
LIN {X 0,Y 481.292,Z 582.634,A -85,B 0,C 180,E1 22525.288,E2 22525.288} C_VEL
LIN {X 0,Y 480.419,Z 601.195,A -85,B 0,C 180,E1 22524.538,E2 22524.538} C_VEL
LIN {X 0,Y 479.428,Z 618.87,A -85,B 0,C 180,E1 22523.604,E2 22523.604} C_VEL
LIN {X 0,Y 478.335,Z 635.688,A -85,B 0,C 180,E1 22522.49,E2 22522.49} C_VEL
LIN {X 0,Y 477.193,Z 651.709,A -85,B 0,C 180,E1 22521.186,E2 22521.186} C_VEL
LIN {X 0,Y 476.057,Z 666.755,A -85,B 0,C 180,E1 22519.7,E2 22519.7} C_VEL
LIN {X 0,Y 474.979,Z 680.816,A -85,B 0,C 180,E1 22518.025,E2 22518.025} C_VEL
LIN {X 0,Y 474.079,Z 692.989,A -85,B 0,C 180,E1 22516.29,E2 22516.29} C_VEL
LIN {X 0,Y 473.281,Z 704.442,A -85,B 0,C 180,E1 22514.31,E2 22514.31} C_VEL
LIN {X 0,Y 472.682,Z 714.316,A -85,B 0,C 180,E1 22512.212,E2 22512.212} C_VEL
LIN {X 0,Y 472.273,Z 722.646,A -85,B 0,C 180,E1 22509.997,E2 22509.997} C_VEL
LIN {X 0,Y 472.049,Z 729.142,A -85,B 0,C 180,E1 22507.791,E2 22507.791} C_VEL
LIN {X 0,Y 471.95,Z 733.915,A -85,B 0,C 180,E1 22505.592,E2 22505.592} C_VEL
LIN {X 0,Y 471.916,Z 737.192,A -85,B 0,C 180,E1 22503.279,E2 22503.279} C_VEL
LIN {X 0,Y 471.916,Z 738.794,A -85,B 0,C 180,E1 22500.971,E2 22500.971} C_VEL
LIN {X 0,Y 471.911,Z 738.735,A -85,B 0,C 180,E1 22498.664,E2 22498.664} C_VEL
LIN {X 0,Y 471.914,Z 737.031,A -85,B 0,C 180,E1 22496.477,E2 22496.477} C_VEL
LIN {X 0,Y 471.953,Z 733.614,A -85,B 0,C 180,E1 22494.163,E2 22494.163} C_VEL
LIN {X 0,Y 472.062,Z 728.762,A -85,B 0,C 180,E1 22491.964,E2 22491.964} C_VEL
LIN {X 0,Y 472.311,Z 721.725,A -85,B 0,C 180,E1 22489.633,E2 22489.633} C_VEL
LIN {X 0,Y 472.711,Z 713.596,A -85,B 0,C 180,E1 22487.54,E2 22487.54} C_VEL
LIN {X 0,Y 473.328,Z 703.509,A -85,B 0,C 180,E1 22485.441,E2 22485.441} C_VEL
LIN {X 0,Y 474.146,Z 691.867,A -85,B 0,C 180,E1 22483.46,E2 22483.46} C_VEL
LIN {X 0,Y 475.156,Z 678.618,A -85,B 0,C 180,E1 22481.6,E2 22481.6} C_VEL
LIN {X 0,Y 476.271,Z 664.265,A -85,B 0,C 180,E1 22479.934,E2 22479.934} C_VEL
LIN {X 0,Y 477.513,Z 648.11,A -85,B 0,C 180,E1 22478.388,E2 22478.388} C_VEL
LIN {X 0,Y 478.711,Z 631.572,A -85,B 0,C 180,E1 22477.088,E2 22477.088} C_VEL
LIN {X 0,Y 479.878,Z 613.747,A -85,B 0,C 180,E1 22475.962,E2 22475.962} C_VEL
LIN {X 0,Y 480.911,Z 595.779,A -85,B 0,C 180,E1 22475.068,E2 22475.068} C_VEL
LIN {X 0,Y 481.785,Z 576.374,A -85,B 0,C 180,E1 22474.348,E2 22474.348} C_VEL
LIN {X 0,Y 482.432,Z 556.759,A -85,B 0,C 180,E1 22473.857,E2 22473.857} C_VEL
LIN {X 0,Y 485.739,Z 361.781,A -85,B 0,C 180,E1 22470.638,E2 22470.638} C_VEL
LIN {X 0,Y 482.407,Z 341.183,A -85,B 0,C 180,E1 22469.997,E2 22469.997} C_VEL
LIN {X 0,Y 484.309,Z 309.352,A -85,B 0,C 180,E1 22467.07,E2 22467.07} C_VEL
LIN {X 0,Y 481.268,Z 300.303,A -85,B 0,C 180,E1 22465.928,E2 22465.928} C_VEL
LIN {X 0,Y 479.033,Z 296.363,A -85,B 0,C 180,E1 22465.344,E2 22465.344} C_VEL
LIN {X 0,Y 472.411,Z 290.224,A -85,B 0,C 180,E1 22464.139,E2 22464.139} C_VEL
LIN {X 0,Y 467.825,Z 285.382,A -85,B 0,C 180,E1 22463.218,E2 22463.218} C_VEL
LIN {X 0,Y 466.245,Z 281.995,A -85,B 0,C 180,E1 22462.715,E2 22462.715} C_VEL
LIN {X 0,Y 465.013,Z 278.744,A -85,B 0,C 180,E1 22462.19,E2 22462.19} C_VEL
LIN {X 0,Y 465.017,Z 278.556,A -85,B 0,C 180,E1 22458.627,E2 22458.627} C_VEL
LIN {X 0,Y 465.012,Z 278.562,A -85,B 0,C 180,E1 22454.975,E2 22454.975} C_VEL
LIN {X 0,Y 465.015,Z 278.563,A -85,B 0,C 180,E1 22451.309,E2 22451.309} C_VEL
LIN {X 0,Y 465.009,Z 278.563,A -85,B 0,C 180,E1 22447.638,E2 22447.638} C_VEL
LIN {X 0,Y 465.01,Z 278.561,A -85,B 0,C 180,E1 22443.903,E2 22443.903} C_VEL
LIN {X 0,Y 465.019,Z 278.553,A -85,B 0,C 180,E1 22440.189,E2 22440.189} C_VEL
LIN {X 0,Y 464.996,Z 278.561,A -85,B 0,C 180,E1 22436.554,E2 22436.554} C_VEL
LIN {X 0,Y 464.979,Z 278.564,A -85,B 0,C 180,E1 22432.906,E2 22432.906} C_VEL
LIN {X 0,Y 464.971,Z 278.565,A -85,B 0,C 180,E1 22429.21,E2 22429.21} C_VEL
LIN {X 0,Y 464.979,Z 278.549,A -85,B 0,C 180,E1 22425.594,E2 22425.594} C_VEL
LIN {X 0,Y 464.982,Z 278.766,A -85,B 0,C 180,E1 22423.113,E2 22423.113} C_VEL
LIN {X 0,Y 466.456,Z 283.117,A -85,B 0,C 180,E1 22422.567,E2 22422.567} C_VEL
LIN {X 0,Y 473.182,Z 302.832,A -85,B 0,C 180,E1 22420.348,E2 22420.348} C_VEL
LIN {X 0,Y 474.745,Z 308.341,A -85,B 0,C 180,E1 22419.762,E2 22419.762} C_VEL
LIN {X 0,Y 473.565,Z 350.556,A -85,B 0,C 180,E1 22416.183,E2 22416.183} C_VEL
LIN {X 0,Y 472.253,Z 392.103,A -85,B 0,C 180,E1 22412.671,E2 22412.671} C_VEL
LIN {X 0,Y 470.814,Z 432.969,A -85,B 0,C 180,E1 22409.21,E2 22409.21} C_VEL
LIN {X 0,Y 469.546,Z 472.848,A -85,B 0,C 180,E1 22405.85,E2 22405.85} C_VEL
LIN {X 0,Y 469.578,Z 476.566,A -85,B 0,C 180,E1 22405.597,E2 22405.597} C_VEL
LIN {X 0,Y 470.822,Z 489.015,A -85,B 0,C 180,E1 22405.34,E2 22405.34} C_VEL
LIN {X 0,Y 469.449,Z 618.878,A -85,B 0,C 180,E1 22403.293,E2 22403.293} C_VEL
LIN {X 0,Y 469.082,Z 634.851,A -85,B 0,C 180,E1 22402.817,E2 22402.817} C_VEL
LIN {X 0,Y 468.512,Z 651.058,A -85,B 0,C 180,E1 22402.089,E2 22402.089} C_VEL
LIN {X 0,Y 467.845,Z 665.454,A -85,B 0,C 180,E1 22401.206,E2 22401.206} C_VEL
LIN {X 0,Y 467.072,Z 679.637,A -85,B 0,C 180,E1 22400.078,E2 22400.078} C_VEL
LIN {X 0,Y 466.353,Z 692.226,A -85,B 0,C 180,E1 22398.813,E2 22398.813} C_VEL
LIN {X 0,Y 465.652,Z 703.866,A -85,B 0,C 180,E1 22397.35,E2 22397.35} C_VEL
LIN {X 0,Y 465.089,Z 713.732,A -85,B 0,C 180,E1 22395.815,E2 22395.815} C_VEL
LIN {X 0,Y 464.603,Z 722.84,A -85,B 0,C 180,E1 22394.012,E2 22394.012} C_VEL
LIN {X 0,Y 464.291,Z 730.112,A -85,B 0,C 180,E1 22392.151,E2 22392.151} C_VEL
LIN {X 0,Y 464.104,Z 735.561,A -85,B 0,C 180,E1 22390.232,E2 22390.232} C_VEL
LIN {X 0,Y 464.018,Z 739.387,A -85,B 0,C 180,E1 22388.237,E2 22388.237} C_VEL
LIN {X 0,Y 463.985,Z 741.358,A -85,B 0,C 180,E1 22386.238,E2 22386.238} C_VEL
LIN {X 0,Y 463.985,Z 741.633,A -85,B 0,C 180,E1 22384.198,E2 22384.198} C_VEL
LIN {X 0,Y 464.005,Z 740.18,A -85,B 0,C 180,E1 22382.263,E2 22382.263} C_VEL
LIN {X 0,Y 464.083,Z 736.734,A -85,B 0,C 180,E1 22380.155,E2 22380.155} C_VEL
LIN {X 0,Y 464.234,Z 731.911,A -85,B 0,C 180,E1 22378.294,E2 22378.294} C_VEL
LIN {X 0,Y 464.513,Z 725.176,A -85,B 0,C 180,E1 22376.411,E2 22376.411} C_VEL
LIN {X 0,Y 464.932,Z 716.977,A -85,B 0,C 180,E1 22374.657,E2 22374.657} C_VEL
LIN {X 0,Y 465.541,Z 706.308,A -85,B 0,C 180,E1 22372.88,E2 22372.88} C_VEL
LIN {X 0,Y 466.222,Z 694.964,A -85,B 0,C 180,E1 22371.388,E2 22371.388} C_VEL
LIN {X 0,Y 466.976,Z 682.126,A -85,B 0,C 180,E1 22370.036,E2 22370.036} C_VEL
LIN {X 0,Y 467.727,Z 668.425,A -85,B 0,C 180,E1 22368.898,E2 22368.898} C_VEL
LIN {X 0,Y 468.461,Z 653.228,A -85,B 0,C 180,E1 22367.921,E2 22367.921} C_VEL
LIN {X 0,Y 469.026,Z 637.742,A -85,B 0,C 180,E1 22367.191,E2 22367.191} C_VEL
LIN {X 0,Y 469.43,Z 621.065,A -85,B 0,C 180,E1 22366.656,E2 22366.656} C_VEL
LIN {X 0,Y 469.75,Z 591.011,A -85,B 0,C 180,E1 22366.144,E2 22366.144} C_VEL
LIN {X 0,Y 470.685,Z 485.447,A -85,B 0,C 180,E1 22364.487,E2 22364.487} C_VEL
LIN {X 0,Y 469.532,Z 475.788,A -85,B 0,C 180,E1 22364.258,E2 22364.258} C_VEL
LIN {X 0,Y 470.835,Z 433.125,A -85,B 0,C 180,E1 22360.689,E2 22360.689} C_VEL
LIN {X 0,Y 472.249,Z 391.324,A -85,B 0,C 180,E1 22357.191,E2 22357.191} C_VEL
LIN {X 0,Y 473.35,Z 347.842,A -85,B 0,C 180,E1 22353.603,E2 22353.603} C_VEL
LIN {X 0,Y 474.148,Z 309.128,A -85,B 0,C 180,E1 22350.405,E2 22350.405} C_VEL
LIN {X 0,Y 473.942,Z 305.321,A -85,B 0,C 180,E1 22350.07,E2 22350.07} C_VEL
LIN {X 0,Y 467.735,Z 286.545,A -85,B 0,C 180,E1 22348.053,E2 22348.053} C_VEL
LIN {X 0,Y 465.04,Z 278.849,A -85,B 0,C 180,E1 22347.152,E2 22347.152} C_VEL
LIN {X 0,Y 465.014,Z 278.559,A -85,B 0,C 180,E1 22345.44,E2 22345.44} C_VEL
LIN {X 0,Y 465.011,Z 278.56,A -85,B 0,C 180,E1 22341.745,E2 22341.745} C_VEL
LIN {X 0,Y 464.981,Z 278.559,A -85,B 0,C 180,E1 22338.12,E2 22338.12} C_VEL
LIN {X 0,Y 464.973,Z 278.563,A -85,B 0,C 180,E1 22334.445,E2 22334.445} C_VEL
LIN {X 0,Y 464.987,Z 278.561,A -85,B 0,C 180,E1 22330.783,E2 22330.783} C_VEL
LIN {X 0,Y 465.019,Z 278.559,A -85,B 0,C 180,E1 22327.164,E2 22327.164} C_VEL
LIN {X 0,Y 465.012,Z 278.562,A -85,B 0,C 180,E1 22323.452,E2 22323.452} C_VEL
LIN {X 0,Y 464.987,Z 278.565,A -85,B 0,C 180,E1 22319.877,E2 22319.877} C_VEL
LIN {X 0,Y 464.977,Z 278.561,A -85,B 0,C 180,E1 22316.302,E2 22316.302} C_VEL
LIN {X 0,Y 464.998,Z 278.559,A -85,B 0,C 180,E1 22312.712,E2 22312.712} C_VEL
LIN {X 0,Y 465.014,Z 278.561,A -85,B 0,C 180,E1 22309.093,E2 22309.093} C_VEL
LIN {X 0,Y 465.016,Z 278.562,A -85,B 0,C 180,E1 22305.361,E2 22305.361} C_VEL
LIN {X 0,Y 464.99,Z 278.565,A -85,B 0,C 180,E1 22301.704,E2 22301.704} C_VEL
LIN {X 0,Y 464.979,Z 278.56,A -85,B 0,C 180,E1 22298.028,E2 22298.028} C_VEL
LIN {X 0,Y 464.992,Z 278.561,A -85,B 0,C 180,E1 22294.393,E2 22294.393} C_VEL
LIN {X 0,Y 465.019,Z 278.557,A -85,B 0,C 180,E1 22290.786,E2 22290.786} C_VEL
LIN {X 0,Y 465.016,Z 278.563,A -85,B 0,C 180,E1 22287.045,E2 22287.045} C_VEL
LIN {X 0,Y 465.004,Z 278.563,A -85,B 0,C 180,E1 22283.321,E2 22283.321} C_VEL
LIN {X 0,Y 464.986,Z 278.563,A -85,B 0,C 180,E1 22279.758,E2 22279.758} C_VEL
LIN {X 0,Y 464.989,Z 278.565,A -85,B 0,C 180,E1 22276.01,E2 22276.01} C_VEL
LIN {X 0,Y 465.01,Z 278.562,A -85,B 0,C 180,E1 22272.464,E2 22272.464} C_VEL
LIN {X 0,Y 465.058,Z 278.859,A -85,B 0,C 180,E1 22270.486,E2 22270.486} C_VEL
LIN {X 0,Y 474.564,Z 302.305,A -85,B 0,C 180,E1 22267.411,E2 22267.411} C_VEL
LIN {X 0,Y 479.76,Z 316.657,A -85,B 0,C 180,E1 22265.716,E2 22265.716} C_VEL
LIN {X 0,Y 482.961,Z 339.639,A -85,B 0,C 180,E1 22264.999,E2 22264.999} C_VEL
LIN {X 0,Y 478.751,Z 545.861,A -85,B 0,C 180,E1 22261.505,E2 22261.505} C_VEL
LIN {X 0,Y 478.071,Z 579.185,A -85,B 0,C 180,E1 22260.922,E2 22260.922} C_VEL
LIN {X 0,Y 477.16,Z 600.106,A -85,B 0,C 180,E1 22260.342,E2 22260.342} C_VEL
LIN {X 0,Y 476.027,Z 620.636,A -85,B 0,C 180,E1 22259.541,E2 22259.541} C_VEL
LIN {X 0,Y 474.706,Z 639.892,A -85,B 0,C 180,E1 22258.561,E2 22258.561} C_VEL
LIN {X 0,Y 473.292,Z 658.653,A -85,B 0,C 180,E1 22257.374,E2 22257.374} C_VEL
LIN {X 0,Y 471.748,Z 677.12,A -85,B 0,C 180,E1 22255.954,E2 22255.954} C_VEL
LIN {X 0,Y 470.177,Z 695.002,A -85,B 0,C 180,E1 22254.297,E2 22254.297} C_VEL
LIN {X 0,Y 468.783,Z 710.825,A -85,B 0,C 180,E1 22252.552,E2 22252.552} C_VEL
LIN {X 0,Y 467.514,Z 725.381,A -85,B 0,C 180,E1 22250.662,E2 22250.662} C_VEL
LIN {X 0,Y 466.423,Z 738.67,A -85,B 0,C 180,E1 22248.625,E2 22248.625} C_VEL
LIN {X 0,Y 465.488,Z 751.127,A -85,B 0,C 180,E1 22246.341,E2 22246.341} C_VEL
LIN {X 0,Y 464.82,Z 761.497,A -85,B 0,C 180,E1 22244.04,E2 22244.04} C_VEL
LIN {X 0,Y 464.368,Z 770.2,A -85,B 0,C 180,E1 22241.676,E2 22241.676} C_VEL
LIN {X 0,Y 464.092,Z 777.478,A -85,B 0,C 180,E1 22239.172,E2 22239.172} C_VEL
LIN {X 0,Y 463.973,Z 782.678,A -85,B 0,C 180,E1 22236.806,E2 22236.806} C_VEL
LIN {X 0,Y 463.918,Z 786.418,A -85,B 0,C 180,E1 22234.325,E2 22234.325} C_VEL
LIN {X 0,Y 463.91,Z 788.349,A -85,B 0,C 180,E1 22231.975,E2 22231.975} C_VEL
LIN {X 0,Y 463.901,Z 788.838,A -85,B 0,C 180,E1 22229.505,E2 22229.505} C_VEL
LIN {X 0,Y 463.908,Z 787.729,A -85,B 0,C 180,E1 22227.034,E2 22227.034} C_VEL
LIN {X 0,Y 463.926,Z 784.921,A -85,B 0,C 180,E1 22224.557,E2 22224.557} C_VEL
LIN {X 0,Y 464.015,Z 780.63,A -85,B 0,C 180,E1 22222.197,E2 22222.197} C_VEL
LIN {X 0,Y 464.202,Z 774.354,A -85,B 0,C 180,E1 22219.7,E2 22219.7} C_VEL
LIN {X 0,Y 464.53,Z 766.554,A -85,B 0,C 180,E1 22217.316,E2 22217.316} C_VEL
LIN {X 0,Y 465.051,Z 757.327,A -85,B 0,C 180,E1 22215.047,E2 22215.047} C_VEL
LIN {X 0,Y 465.784,Z 745.968,A -85,B 0,C 180,E1 22212.767,E2 22212.767} C_VEL
LIN {X 0,Y 466.676,Z 733.824,A -85,B 0,C 180,E1 22210.733,E2 22210.733} C_VEL
LIN {X 0,Y 467.804,Z 719.357,A -85,B 0,C 180,E1 22208.693,E2 22208.693} C_VEL
LIN {X 0,Y 469.049,Z 703.761,A -85,B 0,C 180,E1 22206.844,E2 22206.844} C_VEL
LIN {X 0,Y 470.382,Z 687.086,A -85,B 0,C 180,E1 22205.181,E2 22205.181} C_VEL
LIN {X 0,Y 471.67,Z 670.168,A -85,B 0,C 180,E1 22203.762,E2 22203.762} C_VEL
LIN {X 0,Y 473.009,Z 650.857,A -85,B 0,C 180,E1 22202.423,E2 22202.423} C_VEL
LIN {X 0,Y 474.238,Z 631.347,A -85,B 0,C 180,E1 22201.33,E2 22201.33} C_VEL
LIN {X 0,Y 475.289,Z 611.052,A -85,B 0,C 180,E1 22200.435,E2 22200.435} C_VEL
LIN {X 0,Y 476.177,Z 590.629,A -85,B 0,C 180,E1 22199.764,E2 22199.764} C_VEL
LIN {X 0,Y 476.804,Z 569.324,A -85,B 0,C 180,E1 22199.284,E2 22199.284} C_VEL
LIN {X 0,Y 478.808,Z 448.931,A -85,B 0,C 180,E1 22197.275,E2 22197.275} C_VEL
LIN {X 0,Y 481.529,Z 349.387,A -85,B 0,C 180,E1 22195.413,E2 22195.413} C_VEL
LIN {X 0,Y 481.755,Z 336.867,A -85,B 0,C 180,E1 22195.143,E2 22195.143} C_VEL
LIN {X 0,Y 479.668,Z 320.237,A -85,B 0,C 180,E1 22194.548,E2 22194.548} C_VEL
LIN {X 0,Y 479.84,Z 315.899,A -85,B 0,C 180,E1 22194.151,E2 22194.151} C_VEL
LIN {X 0,Y 476.154,Z 303.9,A -85,B 0,C 180,E1 22192.485,E2 22192.485} C_VEL
LIN {X 0,Y 472.733,Z 294.953,A -85,B 0,C 180,E1 22190.916,E2 22190.916} C_VEL
LIN {X 0,Y 470.866,Z 290.962,A -85,B 0,C 180,E1 22190.046,E2 22190.046} C_VEL
LIN {X 0,Y 469.248,Z 287.348,A -85,B 0,C 180,E1 22189.149,E2 22189.149} C_VEL
LIN {X 0,Y 467.388,Z 283.398,A -85,B 0,C 180,E1 22187.929,E2 22187.929} C_VEL
LIN {X 0,Y 465.308,Z 280.047,A -85,B 0,C 180,E1 22186.217,E2 22186.217} C_VEL
LIN {X 0,Y 465.034,Z 278.718,A -85,B 0,C 180,E1 22185.07,E2 22185.07} C_VEL
LIN {X 0,Y 465.049,Z 278.954,A -85,B 0,C 180,E1 22182.666,E2 22182.666} C_VEL
LIN {X 0,Y 466.072,Z 281.646,A -85,B 0,C 180,E1 22181.03,E2 22181.03} C_VEL
LIN {X 0,Y 467.702,Z 284.057,A -85,B 0,C 180,E1 22179.871,E2 22179.871} C_VEL
LIN {X 0,Y 469.858,Z 288.793,A -85,B 0,C 180,E1 22178.416,E2 22178.416} C_VEL
LIN {X 0,Y 471.799,Z 293.272,A -85,B 0,C 180,E1 22177.308,E2 22177.308} C_VEL
LIN {X 0,Y 475.156,Z 301.73,A -85,B 0,C 180,E1 22175.579,E2 22175.579} C_VEL
LIN {X 0,Y 478.806,Z 313.207,A -85,B 0,C 180,E1 22173.688,E2 22173.688} C_VEL
LIN {X 0,Y 479.261,Z 315.658,A -85,B 0,C 180,E1 22173.348,E2 22173.348} C_VEL
LIN {X 0,Y 476.918,Z 339.639,A -85,B 0,C 180,E1 22170.989,E2 22170.989} C_VEL
LIN {X 0,Y 480.174,Z 361.469,A -85,B 0,C 180,E1 22170.101,E2 22170.101} C_VEL
LIN {X 0,Y 480.378,Z 366.22,A -85,B 0,C 180,E1 22169.965,E2 22169.965} C_VEL
LIN {X 0,Y 477.019,Z 460.537,A -85,B 0,C 180,E1 22168.102,E2 22168.102} C_VEL
LIN {X 0,Y 474.641,Z 563.657,A -85,B 0,C 180,E1 22166.218,E2 22166.218} C_VEL
LIN {X 0,Y 473.877,Z 583.372,A -85,B 0,C 180,E1 22165.638,E2 22165.638} C_VEL
LIN {X 0,Y 472.956,Z 601.758,A -85,B 0,C 180,E1 22164.878,E2 22164.878} C_VEL
LIN {X 0,Y 471.847,Z 620.292,A -85,B 0,C 180,E1 22163.874,E2 22163.874} C_VEL
LIN {X 0,Y 470.644,Z 637.749,A -85,B 0,C 180,E1 22162.68,E2 22162.68} C_VEL
LIN {X 0,Y 469.401,Z 654.23,A -85,B 0,C 180,E1 22161.289,E2 22161.289} C_VEL
LIN {X 0,Y 468.177,Z 669.503,A -85,B 0,C 180,E1 22159.72,E2 22159.72} C_VEL
LIN {X 0,Y 467.107,Z 682.742,A -85,B 0,C 180,E1 22158.082,E2 22158.082} C_VEL
LIN {X 0,Y 466.111,Z 695.456,A -85,B 0,C 180,E1 22156.192,E2 22156.192} C_VEL
LIN {X 0,Y 465.303,Z 706.599,A -85,B 0,C 180,E1 22154.179,E2 22154.179} C_VEL
LIN {X 0,Y 464.7,Z 716.19,A -85,B 0,C 180,E1 22152.046,E2 22152.046} C_VEL
LIN {X 0,Y 464.305,Z 723.807,A -85,B 0,C 180,E1 22149.92,E2 22149.92} C_VEL
LIN {X 0,Y 464.061,Z 730.154,A -85,B 0,C 180,E1 22147.642,E2 22147.642} C_VEL
LIN {X 0,Y 463.956,Z 734.835,A -85,B 0,C 180,E1 22145.317,E2 22145.317} C_VEL
LIN {X 0,Y 463.918,Z 737.769,A -85,B 0,C 180,E1 22142.965,E2 22142.965} C_VEL
LIN {X 0,Y 463.913,Z 739.024,A -85,B 0,C 180,E1 22140.617,E2 22140.617} C_VEL
LIN {X 0,Y 463.909,Z 738.679,A -85,B 0,C 180,E1 22138.27,E2 22138.27} C_VEL
LIN {X 0,Y 463.924,Z 736.7,A -85,B 0,C 180,E1 22135.921,E2 22135.921} C_VEL
LIN {X 0,Y 463.984,Z 732.925,A -85,B 0,C 180,E1 22133.566,E2 22133.566} C_VEL
LIN {X 0,Y 464.132,Z 727.681,A -85,B 0,C 180,E1 22131.326,E2 22131.326} C_VEL
LIN {X 0,Y 464.44,Z 720.672,A -85,B 0,C 180,E1 22129.079,E2 22129.079} C_VEL
LIN {X 0,Y 464.918,Z 712.234,A -85,B 0,C 180,E1 22126.949,E2 22126.949} C_VEL
LIN {X 0,Y 465.629,Z 701.682,A -85,B 0,C 180,E1 22124.812,E2 22124.812} C_VEL
LIN {X 0,Y 466.556,Z 689.485,A -85,B 0,C 180,E1 22122.797,E2 22122.797} C_VEL
LIN {X 0,Y 467.64,Z 676.063,A -85,B 0,C 180,E1 22120.97,E2 22120.97} C_VEL
LIN {X 0,Y 468.845,Z 661.674,A -85,B 0,C 180,E1 22119.332,E2 22119.332} C_VEL
LIN {X 0,Y 470.132,Z 645.791,A -85,B 0,C 180,E1 22117.838,E2 22117.838} C_VEL
LIN {X 0,Y 471.459,Z 628.384,A -85,B 0,C 180,E1 22116.502,E2 22116.502} C_VEL
LIN {X 0,Y 472.634,Z 611.107,A -85,B 0,C 180,E1 22115.436,E2 22115.436} C_VEL
LIN {X 0,Y 473.734,Z 592.303,A -85,B 0,C 180,E1 22114.53,E2 22114.53} C_VEL
LIN {X 0,Y 474.625,Z 573.24,A -85,B 0,C 180,E1 22113.854,E2 22113.854} C_VEL
LIN {X 0,Y 475.261,Z 553.681,A -85,B 0,C 180,E1 22113.392,E2 22113.392} C_VEL
LIN {X 0,Y 478.82,Z 362.881,A -85,B 0,C 180,E1 22110.165,E2 22110.165} C_VEL
LIN {X 0,Y 475.289,Z 340.988,A -85,B 0,C 180,E1 22109.466,E2 22109.466} C_VEL
LIN {X 0,Y 477.161,Z 312.369,A -85,B 0,C 180,E1 22106.797,E2 22106.797} C_VEL
LIN {X 0,Y 470.474,Z 293.202,A -85,B 0,C 180,E1 22104.277,E2 22104.277} C_VEL
LIN {X 0,Y 466.245,Z 281.995,A -85,B 0,C 180,E1 22102.715,E2 22102.715} C_VEL
LIN {X 0,Y 465.187,Z 279.902,A -85,B 0,C 180,E1 22102.287,E2 22102.287} C_VEL
LIN {X 0,Y 463.248,Z 278.89,A -85,B 0,C 180,E1 22101.61,E2 22101.61} C_VEL
LIN {X 0,Y 458.095,Z 279.463,A -85,B 0,C 180,E1 22099.568,E2 22099.568} C_VEL
LIN {X 0,Y 457.07,Z 279.544,A -85,B 0,C 180,E1 22098.475,E2 22098.475} C_VEL
LIN {X 0,Y 457.075,Z 279.552,A -85,B 0,C 180,E1 22094.781,E2 22094.781} C_VEL
LIN {X 0,Y 457.07,Z 279.552,A -85,B 0,C 180,E1 22091,E2 22091} C_VEL
LIN {X 0,Y 457.071,Z 279.553,A -85,B 0,C 180,E1 22087.298,E2 22087.298} C_VEL
LIN {X 0,Y 457.075,Z 279.553,A -85,B 0,C 180,E1 22083.545,E2 22083.545} C_VEL
LIN {X 0,Y 457.076,Z 279.537,A -85,B 0,C 180,E1 22079.774,E2 22079.774} C_VEL
LIN {X 0,Y 457.077,Z 279.547,A -85,B 0,C 180,E1 22076.085,E2 22076.085} C_VEL
LIN {X 0,Y 457.063,Z 279.552,A -85,B 0,C 180,E1 22072.374,E2 22072.374} C_VEL
LIN {X 0,Y 457.034,Z 279.551,A -85,B 0,C 180,E1 22068.761,E2 22068.761} C_VEL
LIN {X 0,Y 457.015,Z 279.526,A -85,B 0,C 180,E1 22065.092,E2 22065.092} C_VEL
LIN {X 0,Y 457.061,Z 279.687,A -85,B 0,C 180,E1 22063.667,E2 22063.667} C_VEL
LIN {X 0,Y 457.527,Z 281.498,A -85,B 0,C 180,E1 22063.395,E2 22063.395} C_VEL
LIN {X 0,Y 464.169,Z 299.981,A -85,B 0,C 180,E1 22061.243,E2 22061.243} C_VEL
LIN {X 0,Y 467.468,Z 310.94,A -85,B 0,C 180,E1 22060.04,E2 22060.04} C_VEL
LIN {X 0,Y 466.22,Z 351.998,A -85,B 0,C 180,E1 22056.528,E2 22056.528} C_VEL
LIN {X 0,Y 464.811,Z 393.857,A -85,B 0,C 180,E1 22052.961,E2 22052.961} C_VEL
LIN {X 0,Y 463.265,Z 435.826,A -85,B 0,C 180,E1 22049.383,E2 22049.383} C_VEL
LIN {X 0,Y 461.963,Z 476.377,A -85,B 0,C 180,E1 22045.961,E2 22045.961} C_VEL
LIN {X 0,Y 463.322,Z 489.694,A -85,B 0,C 180,E1 22045.675,E2 22045.675} C_VEL
LIN {X 0,Y 461.853,Z 619.179,A -85,B 0,C 180,E1 22043.6,E2 22043.6} C_VEL
LIN {X 0,Y 461.468,Z 635.14,A -85,B 0,C 180,E1 22043.118,E2 22043.118} C_VEL
LIN {X 0,Y 460.877,Z 651.033,A -85,B 0,C 180,E1 22042.397,E2 22042.397} C_VEL
LIN {X 0,Y 460.175,Z 665.469,A -85,B 0,C 180,E1 22041.505,E2 22041.505} C_VEL
LIN {X 0,Y 459.346,Z 679.799,A -85,B 0,C 180,E1 22040.353,E2 22040.353} C_VEL
LIN {X 0,Y 458.573,Z 692.45,A -85,B 0,C 180,E1 22039.067,E2 22039.067} C_VEL
LIN {X 0,Y 457.788,Z 704.66,A -85,B 0,C 180,E1 22037.503,E2 22037.503} C_VEL
LIN {X 0,Y 457.187,Z 714.376,A -85,B 0,C 180,E1 22035.952,E2 22035.952} C_VEL
LIN {X 0,Y 456.667,Z 723.439,A -85,B 0,C 180,E1 22034.118,E2 22034.118} C_VEL
LIN {X 0,Y 456.336,Z 730.507,A -85,B 0,C 180,E1 22032.27,E2 22032.27} C_VEL
LIN {X 0,Y 456.125,Z 736.064,A -85,B 0,C 180,E1 22030.272,E2 22030.272} C_VEL
LIN {X 0,Y 456.031,Z 739.827,A -85,B 0,C 180,E1 22028.253,E2 22028.253} C_VEL
LIN {X 0,Y 455.995,Z 741.824,A -85,B 0,C 180,E1 22026.116,E2 22026.116} C_VEL
LIN {X 0,Y 455.995,Z 742.011,A -85,B 0,C 180,E1 22024.131,E2 22024.131} C_VEL
LIN {X 0,Y 456.022,Z 740.332,A -85,B 0,C 180,E1 22022.019,E2 22022.019} C_VEL
LIN {X 0,Y 456.113,Z 736.959,A -85,B 0,C 180,E1 22019.986,E2 22019.986} C_VEL
LIN {X 0,Y 456.296,Z 731.683,A -85,B 0,C 180,E1 22017.978,E2 22017.978} C_VEL
LIN {X 0,Y 456.625,Z 724.766,A -85,B 0,C 180,E1 22016.059,E2 22016.059} C_VEL
LIN {X 0,Y 457.111,Z 716.113,A -85,B 0,C 180,E1 22014.244,E2 22014.244} C_VEL
LIN {X 0,Y 457.756,Z 705.839,A -85,B 0,C 180,E1 22012.54,E2 22012.54} C_VEL
LIN {X 0,Y 458.507,Z 694.154,A -85,B 0,C 180,E1 22011.012,E2 22011.012} C_VEL
LIN {X 0,Y 459.279,Z 681.898,A -85,B 0,C 180,E1 22009.719,E2 22009.719} C_VEL
LIN {X 0,Y 460.074,Z 668.123,A -85,B 0,C 180,E1 22008.572,E2 22008.572} C_VEL
LIN {X 0,Y 460.816,Z 653.687,A -85,B 0,C 180,E1 22007.635,E2 22007.635} C_VEL
LIN {X 0,Y 461.416,Z 638.184,A -85,B 0,C 180,E1 22006.892,E2 22006.892} C_VEL
LIN {X 0,Y 461.845,Z 621.52,A -85,B 0,C 180,E1 22006.349,E2 22006.349} C_VEL
LIN {X 0,Y 462.178,Z 592.418,A -85,B 0,C 180,E1 22005.842,E2 22005.842} C_VEL
LIN {X 0,Y 463.21,Z 486.346,A -85,B 0,C 180,E1 22004.15,E2 22004.15} C_VEL
LIN {X 0,Y 462.002,Z 475.995,A -85,B 0,C 180,E1 22003.893,E2 22003.893} C_VEL
LIN {X 0,Y 463.404,Z 432.873,A -85,B 0,C 180,E1 22000.249,E2 22000.249} C_VEL
LIN {X 0,Y 464.813,Z 391.796,A -85,B 0,C 180,E1 21996.805,E2 21996.805} C_VEL
LIN {X 0,Y 465.885,Z 354.564,A -85,B 0,C 180,E1 21993.689,E2 21993.689} C_VEL
LIN {X 0,Y 466.852,Z 313.786,A -85,B 0,C 180,E1 21990.29,E2 21990.29} C_VEL
LIN {X 0,Y 466.736,Z 308.144,A -85,B 0,C 180,E1 21989.802,E2 21989.802} C_VEL
LIN {X 0,Y 460.194,Z 288.341,A -85,B 0,C 180,E1 21987.638,E2 21987.638} C_VEL
LIN {X 0,Y 457.078,Z 279.857,A -85,B 0,C 180,E1 21986.627,E2 21986.627} C_VEL
LIN {X 0,Y 457.067,Z 279.55,A -85,B 0,C 180,E1 21985.251,E2 21985.251} C_VEL
LIN {X 0,Y 457.08,Z 279.546,A -85,B 0,C 180,E1 21981.562,E2 21981.562} C_VEL
LIN {X 0,Y 457.058,Z 279.548,A -85,B 0,C 180,E1 21977.835,E2 21977.835} C_VEL
LIN {X 0,Y 457.039,Z 279.553,A -85,B 0,C 180,E1 21974.184,E2 21974.184} C_VEL
LIN {X 0,Y 457.037,Z 279.551,A -85,B 0,C 180,E1 21970.462,E2 21970.462} C_VEL
LIN {X 0,Y 457.051,Z 279.549,A -85,B 0,C 180,E1 21966.785,E2 21966.785} C_VEL
LIN {X 0,Y 457.073,Z 279.551,A -85,B 0,C 180,E1 21963.135,E2 21963.135} C_VEL
LIN {X 0,Y 457.081,Z 279.548,A -85,B 0,C 180,E1 21959.374,E2 21959.374} C_VEL
LIN {X 0,Y 457.062,Z 279.55,A -85,B 0,C 180,E1 21955.609,E2 21955.609} C_VEL
LIN {X 0,Y 457.042,Z 279.552,A -85,B 0,C 180,E1 21951.952,E2 21951.952} C_VEL
LIN {X 0,Y 457.04,Z 279.551,A -85,B 0,C 180,E1 21948.261,E2 21948.261} C_VEL
LIN {X 0,Y 457.06,Z 279.545,A -85,B 0,C 180,E1 21944.651,E2 21944.651} C_VEL
LIN {X 0,Y 457.077,Z 279.547,A -85,B 0,C 180,E1 21940.978,E2 21940.978} C_VEL
LIN {X 0,Y 457.082,Z 279.55,A -85,B 0,C 180,E1 21937.221,E2 21937.221} C_VEL
LIN {X 0,Y 457.063,Z 279.554,A -85,B 0,C 180,E1 21933.467,E2 21933.467} C_VEL
LIN {X 0,Y 457.046,Z 279.549,A -85,B 0,C 180,E1 21929.936,E2 21929.936} C_VEL
LIN {X 0,Y 457.051,Z 279.549,A -85,B 0,C 180,E1 21926.229,E2 21926.229} C_VEL
LIN {X 0,Y 457.07,Z 279.548,A -85,B 0,C 180,E1 21922.546,E2 21922.546} C_VEL
LIN {X 0,Y 457.079,Z 279.549,A -85,B 0,C 180,E1 21918.804,E2 21918.804} C_VEL
LIN {X 0,Y 457.073,Z 279.552,A -85,B 0,C 180,E1 21915.044,E2 21915.044} C_VEL
LIN {X 0,Y 457.07,Z 279.628,A -85,B 0,C 180,E1 21911.346,E2 21911.346} C_VEL
LIN {X 0,Y 457.159,Z 280.08,A -85,B 0,C 180,E1 21911.141,E2 21911.141} C_VEL
LIN {X 0,Y 466.829,Z 303.55,A -85,B 0,C 180,E1 21907.984,E2 21907.984} C_VEL
LIN {X 0,Y 472.12,Z 317.423,A -85,B 0,C 180,E1 21906.31,E2 21906.31} C_VEL
LIN {X 0,Y 473.387,Z 320.574,A -85,B 0,C 180,E1 21906.129,E2 21906.129} C_VEL
LIN {X 0,Y 476.224,Z 340.889,A -85,B 0,C 180,E1 21905.502,E2 21905.502} C_VEL
LIN {X 0,Y 471.82,Z 539.098,A -85,B 0,C 180,E1 21902.075,E2 21902.075} C_VEL
LIN {X 0,Y 470.935,Z 578.935,A -85,B 0,C 180,E1 21901.367,E2 21901.367} C_VEL
LIN {X 0,Y 469.987,Z 599.723,A -85,B 0,C 180,E1 21900.784,E2 21900.784} C_VEL
LIN {X 0,Y 468.786,Z 620.058,A -85,B 0,C 180,E1 21899.981,E2 21899.981} C_VEL
LIN {X 0,Y 467.408,Z 639.187,A -85,B 0,C 180,E1 21898.998,E2 21898.998} C_VEL
LIN {X 0,Y 465.933,Z 657.562,A -85,B 0,C 180,E1 21897.828,E2 21897.828} C_VEL
LIN {X 0,Y 464.276,Z 676.292,A -85,B 0,C 180,E1 21896.377,E2 21896.377} C_VEL
LIN {X 0,Y 462.695,Z 693.408,A -85,B 0,C 180,E1 21894.784,E2 21894.784} C_VEL
LIN {X 0,Y 461.202,Z 709.266,A -85,B 0,C 180,E1 21893.034,E2 21893.034} C_VEL
LIN {X 0,Y 459.837,Z 723.952,A -85,B 0,C 180,E1 21891.124,E2 21891.124} C_VEL
LIN {X 0,Y 458.599,Z 737.959,A -85,B 0,C 180,E1 21888.955,E2 21888.955} C_VEL
LIN {X 0,Y 457.644,Z 749.833,A -85,B 0,C 180,E1 21886.76,E2 21886.76} C_VEL
LIN {X 0,Y 456.955,Z 759.754,A -85,B 0,C 180,E1 21884.572,E2 21884.572} C_VEL
LIN {X 0,Y 456.438,Z 768.846,A -85,B 0,C 180,E1 21882.138,E2 21882.138} C_VEL
LIN {X 0,Y 456.143,Z 776.063,A -85,B 0,C 180,E1 21879.716,E2 21879.716} C_VEL
LIN {X 0,Y 455.979,Z 781.782,A -85,B 0,C 180,E1 21877.179,E2 21877.179} C_VEL
LIN {X 0,Y 455.93,Z 785.491,A -85,B 0,C 180,E1 21874.779,E2 21874.779} C_VEL
LIN {X 0,Y 455.918,Z 787.785,A -85,B 0,C 180,E1 21872.261,E2 21872.261} C_VEL
LIN {X 0,Y 455.917,Z 788.456,A -85,B 0,C 180,E1 21869.747,E2 21869.747} C_VEL
LIN {X 0,Y 455.92,Z 787.476,A -85,B 0,C 180,E1 21867.233,E2 21867.233} C_VEL
LIN {X 0,Y 455.931,Z 784.78,A -85,B 0,C 180,E1 21864.714,E2 21864.714} C_VEL
LIN {X 0,Y 456.02,Z 780.371,A -85,B 0,C 180,E1 21862.186,E2 21862.186} C_VEL
LIN {X 0,Y 456.208,Z 774.127,A -85,B 0,C 180,E1 21859.645,E2 21859.645} C_VEL
LIN {X 0,Y 456.546,Z 766.348,A -85,B 0,C 180,E1 21857.22,E2 21857.22} C_VEL
LIN {X 0,Y 457.087,Z 757.112,A -85,B 0,C 180,E1 21854.91,E2 21854.91} C_VEL
LIN {X 0,Y 457.844,Z 745.898,A -85,B 0,C 180,E1 21852.618,E2 21852.618} C_VEL
LIN {X 0,Y 458.789,Z 733.6,A -85,B 0,C 180,E1 21850.521,E2 21850.521} C_VEL
LIN {X 0,Y 459.975,Z 719.116,A -85,B 0,C 180,E1 21848.446,E2 21848.446} C_VEL
LIN {X 0,Y 461.275,Z 703.592,A -85,B 0,C 180,E1 21846.577,E2 21846.577} C_VEL
LIN {X 0,Y 462.631,Z 687.442,A -85,B 0,C 180,E1 21844.937,E2 21844.937} C_VEL
LIN {X 0,Y 464.041,Z 669.844,A -85,B 0,C 180,E1 21843.435,E2 21843.435} C_VEL
LIN {X 0,Y 465.46,Z 650.552,A -85,B 0,C 180,E1 21842.076,E2 21842.076} C_VEL
LIN {X 0,Y 466.817,Z 630.017,A -85,B 0,C 180,E1 21840.912,E2 21840.912} C_VEL
LIN {X 0,Y 467.961,Z 609.395,A -85,B 0,C 180,E1 21840.001,E2 21840.001} C_VEL
LIN {X 0,Y 468.92,Z 587.704,A -85,B 0,C 180,E1 21839.295,E2 21839.295} C_VEL
LIN {X 0,Y 469.574,Z 565.867,A -85,B 0,C 180,E1 21838.825,E2 21838.825} C_VEL
LIN {X 0,Y 471.545,Z 459.985,A -85,B 0,C 180,E1 21837.005,E2 21837.005} C_VEL
LIN {X 0,Y 474.41,Z 365.404,A -85,B 0,C 180,E1 21835.182,E2 21835.182} C_VEL
LIN {X 0,Y 475.268,Z 338.331,A -85,B 0,C 180,E1 21834.604,E2 21834.604} C_VEL
LIN {X 0,Y 473.244,Z 320.921,A -85,B 0,C 180,E1 21833.936,E2 21833.936} C_VEL
LIN {X 0,Y 473.057,Z 318.848,A -85,B 0,C 180,E1 21833.713,E2 21833.713} C_VEL
LIN {X 0,Y 469.658,Z 307.442,A -85,B 0,C 180,E1 21832.029,E2 21832.029} C_VEL
LIN {X 0,Y 466.533,Z 299.194,A -85,B 0,C 180,E1 21830.466,E2 21830.466} C_VEL
LIN {X 0,Y 463.899,Z 293.142,A -85,B 0,C 180,E1 21828.97,E2 21828.97} C_VEL
LIN {X 0,Y 462.143,Z 289.325,A -85,B 0,C 180,E1 21827.711,E2 21827.711} C_VEL
LIN {X 0,Y 460.365,Z 286.081,A -85,B 0,C 180,E1 21825.963,E2 21825.963} C_VEL
LIN {X 0,Y 459.937,Z 284.857,A -85,B 0,C 180,E1 21824.776,E2 21824.776} C_VEL
LIN {X 0,Y 460.05,Z 284.988,A -85,B 0,C 180,E1 21823.034,E2 21823.034} C_VEL
LIN {X 0,Y 460.892,Z 287.554,A -85,B 0,C 180,E1 21821.261,E2 21821.261} C_VEL
LIN {X 0,Y 462.508,Z 290.241,A -85,B 0,C 180,E1 21819.945,E2 21819.945} C_VEL
LIN {X 0,Y 464.521,Z 294.942,A -85,B 0,C 180,E1 21818.466,E2 21818.466} C_VEL
LIN {X 0,Y 467.004,Z 300.757,A -85,B 0,C 180,E1 21817.003,E2 21817.003} C_VEL
LIN {X 0,Y 470.189,Z 309.996,A -85,B 0,C 180,E1 21815.189,E2 21815.189} C_VEL
LIN {X 0,Y 472.686,Z 318.668,A -85,B 0,C 180,E1 21813.766,E2 21813.766} C_VEL
LIN {X 0,Y 470.415,Z 339.223,A -85,B 0,C 180,E1 21811.694,E2 21811.694} C_VEL
LIN {X 0,Y 473.455,Z 359.975,A -85,B 0,C 180,E1 21810.773,E2 21810.773} C_VEL
LIN {X 0,Y 473.986,Z 366.788,A -85,B 0,C 180,E1 21810.538,E2 21810.538} C_VEL
LIN {X 0,Y 470.032,Z 462.753,A -85,B 0,C 180,E1 21808.548,E2 21808.548} C_VEL
LIN {X 0,Y 467.328,Z 564.491,A -85,B 0,C 180,E1 21806.604,E2 21806.604} C_VEL
LIN {X 0,Y 466.49,Z 584.331,A -85,B 0,C 180,E1 21805.996,E2 21805.996} C_VEL
LIN {X 0,Y 465.449,Z 603.573,A -85,B 0,C 180,E1 21805.172,E2 21805.172} C_VEL
LIN {X 0,Y 464.28,Z 621.738,A -85,B 0,C 180,E1 21804.153,E2 21804.153} C_VEL
LIN {X 0,Y 463.025,Z 638.947,A -85,B 0,C 180,E1 21802.944,E2 21802.944} C_VEL
LIN {X 0,Y 461.725,Z 655.288,A -85,B 0,C 180,E1 21801.533,E2 21801.533} C_VEL
LIN {X 0,Y 460.481,Z 669.969,A -85,B 0,C 180,E1 21799.997,E2 21799.997} C_VEL
LIN {X 0,Y 459.311,Z 683.717,A -85,B 0,C 180,E1 21798.268,E2 21798.268} C_VEL
LIN {X 0,Y 458.262,Z 696.374,A -85,B 0,C 180,E1 21796.347,E2 21796.347} C_VEL
LIN {X 0,Y 457.409,Z 707.461,A -85,B 0,C 180,E1 21794.3,E2 21794.3} C_VEL
LIN {X 0,Y 456.77,Z 717.003,A -85,B 0,C 180,E1 21792.13,E2 21792.13} C_VEL
LIN {X 0,Y 456.351,Z 724.573,A -85,B 0,C 180,E1 21789.967,E2 21789.967} C_VEL
LIN {X 0,Y 456.093,Z 730.779,A -85,B 0,C 180,E1 21787.685,E2 21787.685} C_VEL
LIN {X 0,Y 455.974,Z 735.448,A -85,B 0,C 180,E1 21785.284,E2 21785.284} C_VEL
LIN {X 0,Y 455.931,Z 738.322,A -85,B 0,C 180,E1 21782.891,E2 21782.891} C_VEL
LIN {X 0,Y 455.922,Z 739.49,A -85,B 0,C 180,E1 21780.502,E2 21780.502} C_VEL
LIN {X 0,Y 455.92,Z 739.024,A -85,B 0,C 180,E1 21778.114,E2 21778.114} C_VEL
LIN {X 0,Y 455.939,Z 736.915,A -85,B 0,C 180,E1 21775.724,E2 21775.724} C_VEL
LIN {X 0,Y 456.015,Z 733.052,A -85,B 0,C 180,E1 21773.326,E2 21773.326} C_VEL
LIN {X 0,Y 456.209,Z 727.319,A -85,B 0,C 180,E1 21770.92,E2 21770.92} C_VEL
LIN {X 0,Y 456.557,Z 720.008,A -85,B 0,C 180,E1 21768.632,E2 21768.632} C_VEL
LIN {X 0,Y 457.145,Z 710.687,A -85,B 0,C 180,E1 21766.336,E2 21766.336} C_VEL
LIN {X 0,Y 457.968,Z 699.685,A -85,B 0,C 180,E1 21764.162,E2 21764.162} C_VEL
LIN {X 0,Y 458.995,Z 687.344,A -85,B 0,C 180,E1 21762.167,E2 21762.167} C_VEL
LIN {X 0,Y 460.155,Z 674.019,A -85,B 0,C 180,E1 21760.384,E2 21760.384} C_VEL
LIN {X 0,Y 461.415,Z 659.738,A -85,B 0,C 180,E1 21758.784,E2 21758.784} C_VEL
LIN {X 0,Y 462.762,Z 643.878,A -85,B 0,C 180,E1 21757.309,E2 21757.309} C_VEL
LIN {X 0,Y 464.102,Z 627.202,A -85,B 0,C 180,E1 21756.039,E2 21756.039} C_VEL
LIN {X 0,Y 465.366,Z 609.596,A -85,B 0,C 180,E1 21754.959,E2 21754.959} C_VEL
LIN {X 0,Y 466.447,Z 591.759,A -85,B 0,C 180,E1 21754.103,E2 21754.103} C_VEL
LIN {X 0,Y 467.379,Z 572.839,A -85,B 0,C 180,E1 21753.429,E2 21753.429} C_VEL
LIN {X 0,Y 468.043,Z 553.455,A -85,B 0,C 180,E1 21752.968,E2 21752.968} C_VEL
LIN {X 0,Y 472.044,Z 364.66,A -85,B 0,C 180,E1 21749.699,E2 21749.699} C_VEL
LIN {X 0,Y 468.212,Z 340.667,A -85,B 0,C 180,E1 21748.908,E2 21748.908} C_VEL
LIN {X 0,Y 469.992,Z 315.315,A -85,B 0,C 180,E1 21746.507,E2 21746.507} C_VEL
LIN {X 0,Y 463.477,Z 296.548,A -85,B 0,C 180,E1 21743.998,E2 21743.998} C_VEL
LIN {X 0,Y 457.078,Z 279.761,A -85,B 0,C 180,E1 21741.536,E2 21741.536} C_VEL
LIN {X 0,Y 457.07,Z 279.544,A -85,B 0,C 180,E1 21738.475,E2 21738.475} C_VEL
LIN {X 0,Y 456.059,Z 279.675,A -85,B 0,C 180,E1 21737.51,E2 21737.51} C_VEL
LIN {X 0,Y 449.569,Z 280.487,A -85,B 0,C 180,E1 21734.722,E2 21734.722} C_VEL
LIN {X 0,Y 449.122,Z 280.541,A -85,B 0,C 180,E1 21734.083,E2 21734.083} C_VEL
LIN {X 0,Y 449.137,Z 280.538,A -85,B 0,C 180,E1 21730.378,E2 21730.378} C_VEL
LIN {X 0,Y 449.13,Z 280.537,A -85,B 0,C 180,E1 21726.63,E2 21726.63} C_VEL
LIN {X 0,Y 449.119,Z 280.539,A -85,B 0,C 180,E1 21722.903,E2 21722.903} C_VEL
LIN {X 0,Y 449.114,Z 280.527,A -85,B 0,C 180,E1 21719.181,E2 21719.181} C_VEL
LIN {X 0,Y 449.118,Z 280.528,A -85,B 0,C 180,E1 21715.448,E2 21715.448} C_VEL
LIN {X 0,Y 449.137,Z 280.53,A -85,B 0,C 180,E1 21711.824,E2 21711.824} C_VEL
LIN {X 0,Y 449.133,Z 280.53,A -85,B 0,C 180,E1 21708.027,E2 21708.027} C_VEL
LIN {X 0,Y 449.131,Z 280.608,A -85,B 0,C 180,E1 21704.248,E2 21704.248} C_VEL
LIN {X 0,Y 449.544,Z 282.242,A -85,B 0,C 180,E1 21703.966,E2 21703.966} C_VEL
LIN {X 0,Y 456.659,Z 302.01,A -85,B 0,C 180,E1 21701.622,E2 21701.622} C_VEL
LIN {X 0,Y 460.21,Z 313.576,A -85,B 0,C 180,E1 21700.327,E2 21700.327} C_VEL
LIN {X 0,Y 458.853,Z 354.962,A -85,B 0,C 180,E1 21696.759,E2 21696.759} C_VEL
LIN {X 0,Y 457.35,Z 396.302,A -85,B 0,C 180,E1 21693.197,E2 21693.197} C_VEL
LIN {X 0,Y 455.74,Z 437.908,A -85,B 0,C 180,E1 21689.624,E2 21689.624} C_VEL
LIN {X 0,Y 454.421,Z 476.738,A -85,B 0,C 180,E1 21686.319,E2 21686.319} C_VEL
LIN {X 0,Y 455.836,Z 490.567,A -85,B 0,C 180,E1 21686.018,E2 21686.018} C_VEL
LIN {X 0,Y 454.268,Z 619.633,A -85,B 0,C 180,E1 21683.913,E2 21683.913} C_VEL
LIN {X 0,Y 453.856,Z 635.661,A -85,B 0,C 180,E1 21683.419,E2 21683.419} C_VEL
LIN {X 0,Y 453.255,Z 650.989,A -85,B 0,C 180,E1 21682.714,E2 21682.714} C_VEL
LIN {X 0,Y 452.533,Z 665.232,A -85,B 0,C 180,E1 21681.831,E2 21681.831} C_VEL
LIN {X 0,Y 451.63,Z 679.94,A -85,B 0,C 180,E1 21680.637,E2 21680.637} C_VEL
LIN {X 0,Y 450.841,Z 692.096,A -85,B 0,C 180,E1 21679.394,E2 21679.394} C_VEL
LIN {X 0,Y 450.014,Z 704.083,A -85,B 0,C 180,E1 21677.856,E2 21677.856} C_VEL
LIN {X 0,Y 449.336,Z 714.291,A -85,B 0,C 180,E1 21676.227,E2 21676.227} C_VEL
LIN {X 0,Y 448.765,Z 723.452,A -85,B 0,C 180,E1 21674.362,E2 21674.362} C_VEL
LIN {X 0,Y 448.394,Z 730.619,A -85,B 0,C 180,E1 21672.482,E2 21672.482} C_VEL
LIN {X 0,Y 448.159,Z 736.252,A -85,B 0,C 180,E1 21670.45,E2 21670.45} C_VEL
LIN {X 0,Y 448.048,Z 740.095,A -85,B 0,C 180,E1 21668.396,E2 21668.396} C_VEL
LIN {X 0,Y 448.006,Z 742.118,A -85,B 0,C 180,E1 21666.316,E2 21666.316} C_VEL
LIN {X 0,Y 448.004,Z 742.42,A -85,B 0,C 180,E1 21664.204,E2 21664.204} C_VEL
LIN {X 0,Y 448.031,Z 741.006,A -85,B 0,C 180,E1 21662.2,E2 21662.2} C_VEL
LIN {X 0,Y 448.127,Z 737.586,A -85,B 0,C 180,E1 21660.016,E2 21660.016} C_VEL
LIN {X 0,Y 448.31,Z 732.813,A -85,B 0,C 180,E1 21658.093,E2 21658.093} C_VEL
LIN {X 0,Y 448.644,Z 726.109,A -85,B 0,C 180,E1 21656.143,E2 21656.143} C_VEL
LIN {X 0,Y 449.14,Z 717.93,A -85,B 0,C 180,E1 21654.322,E2 21654.322} C_VEL
LIN {X 0,Y 449.832,Z 707.5,A -85,B 0,C 180,E1 21652.517,E2 21652.517} C_VEL
LIN {X 0,Y 450.573,Z 696.876,A -85,B 0,C 180,E1 21651.045,E2 21651.045} C_VEL
LIN {X 0,Y 451.426,Z 684.129,A -85,B 0,C 180,E1 21649.635,E2 21649.635} C_VEL
LIN {X 0,Y 452.278,Z 670.794,A -85,B 0,C 180,E1 21648.457,E2 21648.457} C_VEL
LIN {X 0,Y 453.084,Z 656.003,A -85,B 0,C 180,E1 21647.45,E2 21647.45} C_VEL
LIN {X 0,Y 453.737,Z 641.285,A -85,B 0,C 180,E1 21646.692,E2 21646.692} C_VEL
LIN {X 0,Y 454.202,Z 625.159,A -85,B 0,C 180,E1 21646.119,E2 21646.119} C_VEL
LIN {X 0,Y 454.475,Z 607.28,A -85,B 0,C 180,E1 21645.746,E2 21645.746} C_VEL
LIN {X 0,Y 455.734,Z 487.115,A -85,B 0,C 180,E1 21643.8,E2 21643.8} C_VEL
LIN {X 0,Y 454.494,Z 476.284,A -85,B 0,C 180,E1 21643.519,E2 21643.519} C_VEL
LIN {X 0,Y 455.937,Z 434.163,A -85,B 0,C 180,E1 21639.929,E2 21639.929} C_VEL
LIN {X 0,Y 457.572,Z 390.761,A -85,B 0,C 180,E1 21636.234,E2 21636.234} C_VEL
LIN {X 0,Y 458.845,Z 346.921,A -85,B 0,C 180,E1 21632.564,E2 21632.564} C_VEL
LIN {X 0,Y 459.697,Z 311.528,A -85,B 0,C 180,E1 21629.587,E2 21629.587} C_VEL
LIN {X 0,Y 453.193,Z 291.764,A -85,B 0,C 180,E1 21627.388,E2 21627.388} C_VEL
LIN {X 0,Y 449.163,Z 280.91,A -85,B 0,C 180,E1 21626.082,E2 21626.082} C_VEL
LIN {X 0,Y 449.136,Z 280.536,A -85,B 0,C 180,E1 21625.587,E2 21625.587} C_VEL
LIN {X 0,Y 449.126,Z 280.539,A -85,B 0,C 180,E1 21621.826,E2 21621.826} C_VEL
LIN {X 0,Y 449.102,Z 280.536,A -85,B 0,C 180,E1 21618.162,E2 21618.162} C_VEL
LIN {X 0,Y 449.096,Z 280.541,A -85,B 0,C 180,E1 21614.433,E2 21614.433} C_VEL
LIN {X 0,Y 449.109,Z 280.539,A -85,B 0,C 180,E1 21610.779,E2 21610.779} C_VEL
LIN {X 0,Y 449.141,Z 280.537,A -85,B 0,C 180,E1 21607.162,E2 21607.162} C_VEL
LIN {X 0,Y 449.134,Z 280.54,A -85,B 0,C 180,E1 21603.446,E2 21603.446} C_VEL
LIN {X 0,Y 449.119,Z 280.544,A -85,B 0,C 180,E1 21599.745,E2 21599.745} C_VEL
LIN {X 0,Y 449.103,Z 280.539,A -85,B 0,C 180,E1 21596.043,E2 21596.043} C_VEL
LIN {X 0,Y 449.102,Z 280.539,A -85,B 0,C 180,E1 21592.324,E2 21592.324} C_VEL
LIN {X 0,Y 449.12,Z 280.538,A -85,B 0,C 180,E1 21588.702,E2 21588.702} C_VEL
LIN {X 0,Y 449.142,Z 280.535,A -85,B 0,C 180,E1 21585.035,E2 21585.035} C_VEL
LIN {X 0,Y 449.134,Z 280.537,A -85,B 0,C 180,E1 21581.303,E2 21581.303} C_VEL
LIN {X 0,Y 449.114,Z 280.538,A -85,B 0,C 180,E1 21577.624,E2 21577.624} C_VEL
LIN {X 0,Y 449.104,Z 280.541,A -85,B 0,C 180,E1 21573.987,E2 21573.987} C_VEL
LIN {X 0,Y 449.11,Z 280.536,A -85,B 0,C 180,E1 21570.234,E2 21570.234} C_VEL
LIN {X 0,Y 449.133,Z 280.537,A -85,B 0,C 180,E1 21566.594,E2 21566.594} C_VEL
LIN {X 0,Y 449.139,Z 280.538,A -85,B 0,C 180,E1 21562.838,E2 21562.838} C_VEL
LIN {X 0,Y 449.139,Z 280.54,A -85,B 0,C 180,E1 21559.119,E2 21559.119} C_VEL
LIN {X 0,Y 449.119,Z 280.541,A -85,B 0,C 180,E1 21555.428,E2 21555.428} C_VEL
LIN {X 0,Y 449.141,Z 280.773,A -85,B 0,C 180,E1 21551.922,E2 21551.922} C_VEL
LIN {X 0,Y 451.649,Z 287.077,A -85,B 0,C 180,E1 21550.983,E2 21550.983} C_VEL
LIN {X 0,Y 460.318,Z 307.995,A -85,B 0,C 180,E1 21548.159,E2 21548.159} C_VEL
LIN {X 0,Y 463.887,Z 317.307,A -85,B 0,C 180,E1 21547.006,E2 21547.006} C_VEL
LIN {X 0,Y 467.002,Z 323.829,A -85,B 0,C 180,E1 21546.588,E2 21546.588} C_VEL
LIN {X 0,Y 469.493,Z 342.184,A -85,B 0,C 180,E1 21546.012,E2 21546.012} C_VEL
LIN {X 0,Y 464.853,Z 535.757,A -85,B 0,C 180,E1 21542.6,E2 21542.6} C_VEL
LIN {X 0,Y 463.81,Z 578.935,A -85,B 0,C 180,E1 21541.815,E2 21541.815} C_VEL
LIN {X 0,Y 462.812,Z 599.678,A -85,B 0,C 180,E1 21541.224,E2 21541.224} C_VEL
LIN {X 0,Y 461.518,Z 620.38,A -85,B 0,C 180,E1 21540.394,E2 21540.394} C_VEL
LIN {X 0,Y 460.009,Z 640.141,A -85,B 0,C 180,E1 21539.356,E2 21539.356} C_VEL
LIN {X 0,Y 458.457,Z 658.206,A -85,B 0,C 180,E1 21538.173,E2 21538.173} C_VEL
LIN {X 0,Y 456.739,Z 676.474,A -85,B 0,C 180,E1 21536.727,E2 21536.727} C_VEL
LIN {X 0,Y 454.965,Z 694.499,A -85,B 0,C 180,E1 21535.006,E2 21535.006} C_VEL
LIN {X 0,Y 453.312,Z 711.029,A -85,B 0,C 180,E1 21533.115,E2 21533.115} C_VEL
LIN {X 0,Y 451.875,Z 725.61,A -85,B 0,C 180,E1 21531.139,E2 21531.139} C_VEL
LIN {X 0,Y 450.656,Z 738.782,A -85,B 0,C 180,E1 21529.033,E2 21529.033} C_VEL
LIN {X 0,Y 449.621,Z 751.154,A -85,B 0,C 180,E1 21526.669,E2 21526.669} C_VEL
LIN {X 0,Y 448.858,Z 761.842,A -85,B 0,C 180,E1 21524.182,E2 21524.182} C_VEL
LIN {X 0,Y 448.37,Z 770.416,A -85,B 0,C 180,E1 21521.707,E2 21521.707} C_VEL
LIN {X 0,Y 448.097,Z 777.147,A -85,B 0,C 180,E1 21519.243,E2 21519.243} C_VEL
LIN {X 0,Y 447.976,Z 782.424,A -85,B 0,C 180,E1 21516.663,E2 21516.663} C_VEL
LIN {X 0,Y 447.934,Z 785.83,A -85,B 0,C 180,E1 21514.223,E2 21514.223} C_VEL
LIN {X 0,Y 447.924,Z 787.706,A -85,B 0,C 180,E1 21511.661,E2 21511.661} C_VEL
LIN {X 0,Y 447.93,Z 787.934,A -85,B 0,C 180,E1 21509.231,E2 21509.231} C_VEL
LIN {X 0,Y 447.924,Z 786.591,A -85,B 0,C 180,E1 21506.671,E2 21506.671} C_VEL
LIN {X 0,Y 447.954,Z 783.781,A -85,B 0,C 180,E1 21504.234,E2 21504.234} C_VEL
LIN {X 0,Y 448.055,Z 779.035,A -85,B 0,C 180,E1 21501.658,E2 21501.658} C_VEL
LIN {X 0,Y 448.26,Z 772.794,A -85,B 0,C 180,E1 21499.2,E2 21499.2} C_VEL
LIN {X 0,Y 448.64,Z 764.715,A -85,B 0,C 180,E1 21496.728,E2 21496.728} C_VEL
LIN {X 0,Y 449.278,Z 754.556,A -85,B 0,C 180,E1 21494.245,E2 21494.245} C_VEL
LIN {X 0,Y 450.13,Z 743.005,A -85,B 0,C 180,E1 21491.933,E2 21491.933} C_VEL
LIN {X 0,Y 451.188,Z 730.06,A -85,B 0,C 180,E1 21489.774,E2 21489.774} C_VEL
LIN {X 0,Y 452.465,Z 715.399,A -85,B 0,C 180,E1 21487.728,E2 21487.728} C_VEL
LIN {X 0,Y 453.839,Z 699.789,A -85,B 0,C 180,E1 21485.897,E2 21485.897} C_VEL
LIN {X 0,Y 455.316,Z 682.894,A -85,B 0,C 180,E1 21484.226,E2 21484.226} C_VEL
LIN {X 0,Y 456.751,Z 665.337,A -85,B 0,C 180,E1 21482.772,E2 21482.772} C_VEL
LIN {X 0,Y 458.24,Z 646.072,A -85,B 0,C 180,E1 21481.454,E2 21481.454} C_VEL
LIN {X 0,Y 459.606,Z 625.931,A -85,B 0,C 180,E1 21480.344,E2 21480.344} C_VEL
LIN {X 0,Y 460.785,Z 605.455,A -85,B 0,C 180,E1 21479.466,E2 21479.466} C_VEL
LIN {X 0,Y 461.742,Z 584.721,A -85,B 0,C 180,E1 21478.812,E2 21478.812} C_VEL
LIN {X 0,Y 462.403,Z 562.319,A -85,B 0,C 180,E1 21478.342,E2 21478.342} C_VEL
LIN {X 0,Y 464.451,Z 466.12,A -85,B 0,C 180,E1 21476.629,E2 21476.629} C_VEL
LIN {X 0,Y 467.579,Z 374.807,A -85,B 0,C 180,E1 21474.801,E2 21474.801} C_VEL
LIN {X 0,Y 468.939,Z 339.731,A -85,B 0,C 180,E1 21474.026,E2 21474.026} C_VEL
LIN {X 0,Y 467.087,Z 323.355,A -85,B 0,C 180,E1 21473.366,E2 21473.366} C_VEL
LIN {X 0,Y 466.104,Z 320.719,A -85,B 0,C 180,E1 21473.083,E2 21473.083} C_VEL
LIN {X 0,Y 463.19,Z 310.793,A -85,B 0,C 180,E1 21471.49,E2 21471.49} C_VEL
LIN {X 0,Y 460.486,Z 303.252,A -85,B 0,C 180,E1 21469.951,E2 21469.951} C_VEL
LIN {X 0,Y 458.316,Z 298.482,A -85,B 0,C 180,E1 21468.621,E2 21468.621} C_VEL
LIN {X 0,Y 456.97,Z 295.312,A -85,B 0,C 180,E1 21467.507,E2 21467.507} C_VEL
LIN {X 0,Y 455.479,Z 292.157,A -85,B 0,C 180,E1 21465.694,E2 21465.694} C_VEL
LIN {X 0,Y 455.145,Z 291.254,A -85,B 0,C 180,E1 21464.621,E2 21464.621} C_VEL
LIN {X 0,Y 455.306,Z 291.516,A -85,B 0,C 180,E1 21462.903,E2 21462.903} C_VEL
LIN {X 0,Y 456.358,Z 294.584,A -85,B 0,C 180,E1 21460.897,E2 21460.897} C_VEL
LIN {X 0,Y 457.325,Z 296.299,A -85,B 0,C 180,E1 21460.073,E2 21460.073} C_VEL
LIN {X 0,Y 458.999,Z 300.428,A -85,B 0,C 180,E1 21458.695,E2 21458.695} C_VEL
LIN {X 0,Y 461.244,Z 306.052,A -85,B 0,C 180,E1 21457.214,E2 21457.214} C_VEL
LIN {X 0,Y 464.121,Z 314.873,A -85,B 0,C 180,E1 21455.416,E2 21455.416} C_VEL
LIN {X 0,Y 466.083,Z 322.779,A -85,B 0,C 180,E1 21454.099,E2 21454.099} C_VEL
LIN {X 0,Y 464.085,Z 338.535,A -85,B 0,C 180,E1 21452.461,E2 21452.461} C_VEL
LIN {X 0,Y 466.875,Z 358.34,A -85,B 0,C 180,E1 21451.507,E2 21451.507} C_VEL
LIN {X 0,Y 467.732,Z 367.877,A -85,B 0,C 180,E1 21451.134,E2 21451.134} C_VEL
LIN {X 0,Y 463.358,Z 459.298,A -85,B 0,C 180,E1 21449.139,E2 21449.139} C_VEL
LIN {X 0,Y 460.584,Z 549.83,A -85,B 0,C 180,E1 21447.351,E2 21447.351} C_VEL
LIN {X 0,Y 459.83,Z 571.487,A -85,B 0,C 180,E1 21446.846,E2 21446.846} C_VEL
LIN {X 0,Y 458.842,Z 591.186,A -85,B 0,C 180,E1 21446.146,E2 21446.146} C_VEL
LIN {X 0,Y 457.656,Z 610.428,A -85,B 0,C 180,E1 21445.215,E2 21445.215} C_VEL
LIN {X 0,Y 456.377,Z 628.154,A -85,B 0,C 180,E1 21444.116,E2 21444.116} C_VEL
LIN {X 0,Y 455.03,Z 644.916,A -85,B 0,C 180,E1 21442.83,E2 21442.83} C_VEL
LIN {X 0,Y 453.711,Z 660.341,A -85,B 0,C 180,E1 21441.39,E2 21441.39} C_VEL
LIN {X 0,Y 452.418,Z 674.823,A -85,B 0,C 180,E1 21439.763,E2 21439.763} C_VEL
LIN {X 0,Y 451.209,Z 688.298,A -85,B 0,C 180,E1 21437.939,E2 21437.939} C_VEL
LIN {X 0,Y 450.168,Z 700.262,A -85,B 0,C 180,E1 21435.986,E2 21435.986} C_VEL
LIN {X 0,Y 449.334,Z 710.752,A -85,B 0,C 180,E1 21433.905,E2 21433.905} C_VEL
LIN {X 0,Y 448.713,Z 719.754,A -85,B 0,C 180,E1 21431.699,E2 21431.699} C_VEL
LIN {X 0,Y 448.319,Z 726.882,A -85,B 0,C 180,E1 21429.499,E2 21429.499} C_VEL
LIN {X 0,Y 448.084,Z 732.617,A -85,B 0,C 180,E1 21427.178,E2 21427.178} C_VEL
LIN {X 0,Y 447.975,Z 736.798,A -85,B 0,C 180,E1 21424.737,E2 21424.737} C_VEL
LIN {X 0,Y 447.941,Z 739.228,A -85,B 0,C 180,E1 21422.302,E2 21422.302} C_VEL
LIN {X 0,Y 447.94,Z 739.996,A -85,B 0,C 180,E1 21419.872,E2 21419.872} C_VEL
LIN {X 0,Y 447.94,Z 739.07,A -85,B 0,C 180,E1 21417.441,E2 21417.441} C_VEL
LIN {X 0,Y 447.974,Z 736.442,A -85,B 0,C 180,E1 21415.006,E2 21415.006} C_VEL
LIN {X 0,Y 448.088,Z 732.064,A -85,B 0,C 180,E1 21412.563,E2 21412.563} C_VEL
LIN {X 0,Y 448.35,Z 725.79,A -85,B 0,C 180,E1 21410.112,E2 21410.112} C_VEL
LIN {X 0,Y 448.796,Z 717.917,A -85,B 0,C 180,E1 21407.781,E2 21407.781} C_VEL
LIN {X 0,Y 449.462,Z 708.514,A -85,B 0,C 180,E1 21405.572,E2 21405.572} C_VEL
LIN {X 0,Y 450.354,Z 697.621,A -85,B 0,C 180,E1 21403.49,E2 21403.49} C_VEL
LIN {X 0,Y 451.46,Z 685.251,A -85,B 0,C 180,E1 21401.536,E2 21401.536} C_VEL
LIN {X 0,Y 452.754,Z 671.351,A -85,B 0,C 180,E1 21399.713,E2 21399.713} C_VEL
LIN {X 0,Y 454.128,Z 656.651,A -85,B 0,C 180,E1 21398.108,E2 21398.108} C_VEL
LIN {X 0,Y 455.557,Z 640.643,A -85,B 0,C 180,E1 21396.661,E2 21396.661} C_VEL
LIN {X 0,Y 456.934,Z 624.078,A -85,B 0,C 180,E1 21395.432,E2 21395.432} C_VEL
LIN {X 0,Y 458.211,Z 606.847,A -85,B 0,C 180,E1 21394.401,E2 21394.401} C_VEL
LIN {X 0,Y 459.404,Z 587.701,A -85,B 0,C 180,E1 21393.519,E2 21393.519} C_VEL
LIN {X 0,Y 460.322,Z 568.448,A -85,B 0,C 180,E1 21392.876,E2 21392.876} C_VEL
LIN {X 0,Y 460.979,Z 547.683,A -85,B 0,C 180,E1 21392.43,E2 21392.43} C_VEL
LIN {X 0,Y 465.162,Z 367.88,A -85,B 0,C 180,E1 21389.245,E2 21389.245} C_VEL
LIN {X 0,Y 464.681,Z 362.556,A -85,B 0,C 180,E1 21389.101,E2 21389.101} C_VEL
LIN {X 0,Y 461.179,Z 340.621,A -85,B 0,C 180,E1 21388.353,E2 21388.353} C_VEL
LIN {X 0,Y 462.937,Z 318.632,A -85,B 0,C 180,E1 21386.257,E2 21386.257} C_VEL
LIN {X 0,Y 456.59,Z 300.164,A -85,B 0,C 180,E1 21383.753,E2 21383.753} C_VEL
LIN {X 0,Y 449.169,Z 280.738,A -85,B 0,C 180,E1 21380.865,E2 21380.865} C_VEL
LIN {X 0,Y 449.133,Z 280.54,A -85,B 0,C 180,E1 21377.234,E2 21377.234} C_VEL
LIN {X 0,Y 449.122,Z 280.541,A -85,B 0,C 180,E1 21374.083,E2 21374.083} C_VEL
LIN {X 0,Y 448.112,Z 280.666,A -85,B 0,C 180,E1 21373.101,E2 21373.101} C_VEL
LIN {X 0,Y 441.609,Z 281.477,A -85,B 0,C 180,E1 21370.262,E2 21370.262} C_VEL
LIN {X 0,Y 441.192,Z 281.529,A -85,B 0,C 180,E1 21369.612,E2 21369.612} C_VEL
LIN {X 0,Y 441.191,Z 281.529,A -85,B 0,C 180,E1 21365.773,E2 21365.773} C_VEL
LIN {X 0,Y 441.198,Z 281.527,A -85,B 0,C 180,E1 21362.027,E2 21362.027} C_VEL
LIN {X 0,Y 441.199,Z 281.519,A -85,B 0,C 180,E1 21358.272,E2 21358.272} C_VEL
LIN {X 0,Y 441.18,Z 281.517,A -85,B 0,C 180,E1 21354.504,E2 21354.504} C_VEL
LIN {X 0,Y 441.158,Z 281.522,A -85,B 0,C 180,E1 21350.846,E2 21350.846} C_VEL
LIN {X 0,Y 441.149,Z 281.531,A -85,B 0,C 180,E1 21347.137,E2 21347.137} C_VEL
LIN {X 0,Y 441.173,Z 281.72,A -85,B 0,C 180,E1 21344.773,E2 21344.773} C_VEL
LIN {X 0,Y 442.32,Z 284.77,A -85,B 0,C 180,E1 21344.332,E2 21344.332} C_VEL
LIN {X 0,Y 450.223,Z 307.11,A -85,B 0,C 180,E1 21341.653,E2 21341.653} C_VEL
LIN {X 0,Y 452.973,Z 316.25,A -85,B 0,C 180,E1 21340.622,E2 21340.622} C_VEL
LIN {X 0,Y 451.506,Z 357.126,A -85,B 0,C 180,E1 21337.061,E2 21337.061} C_VEL
LIN {X 0,Y 449.934,Z 398.081,A -85,B 0,C 180,E1 21333.505,E2 21333.505} C_VEL
LIN {X 0,Y 448.236,Z 439.173,A -85,B 0,C 180,E1 21329.937,E2 21329.937} C_VEL
LIN {X 0,Y 446.887,Z 477.018,A -85,B 0,C 180,E1 21326.691,E2 21326.691} C_VEL
LIN {X 0,Y 448.356,Z 491.357,A -85,B 0,C 180,E1 21326.369,E2 21326.369} C_VEL
LIN {X 0,Y 446.695,Z 620.089,A -85,B 0,C 180,E1 21324.237,E2 21324.237} C_VEL
LIN {X 0,Y 446.261,Z 636.081,A -85,B 0,C 180,E1 21323.735,E2 21323.735} C_VEL
LIN {X 0,Y 445.592,Z 652.169,A -85,B 0,C 180,E1 21322.977,E2 21322.977} C_VEL
LIN {X 0,Y 444.806,Z 666.508,A -85,B 0,C 180,E1 21322.055,E2 21322.055} C_VEL
LIN {X 0,Y 443.877,Z 680.803,A -85,B 0,C 180,E1 21320.864,E2 21320.864} C_VEL
LIN {X 0,Y 442.998,Z 693.41,A -85,B 0,C 180,E1 21319.533,E2 21319.533} C_VEL
LIN {X 0,Y 442.144,Z 705.063,A -85,B 0,C 180,E1 21317.994,E2 21317.994} C_VEL
LIN {X 0,Y 441.429,Z 715.121,A -85,B 0,C 180,E1 21316.341,E2 21316.341} C_VEL
LIN {X 0,Y 440.834,Z 724.039,A -85,B 0,C 180,E1 21314.478,E2 21314.478} C_VEL
LIN {X 0,Y 440.434,Z 731.159,A -85,B 0,C 180,E1 21312.564,E2 21312.564} C_VEL
